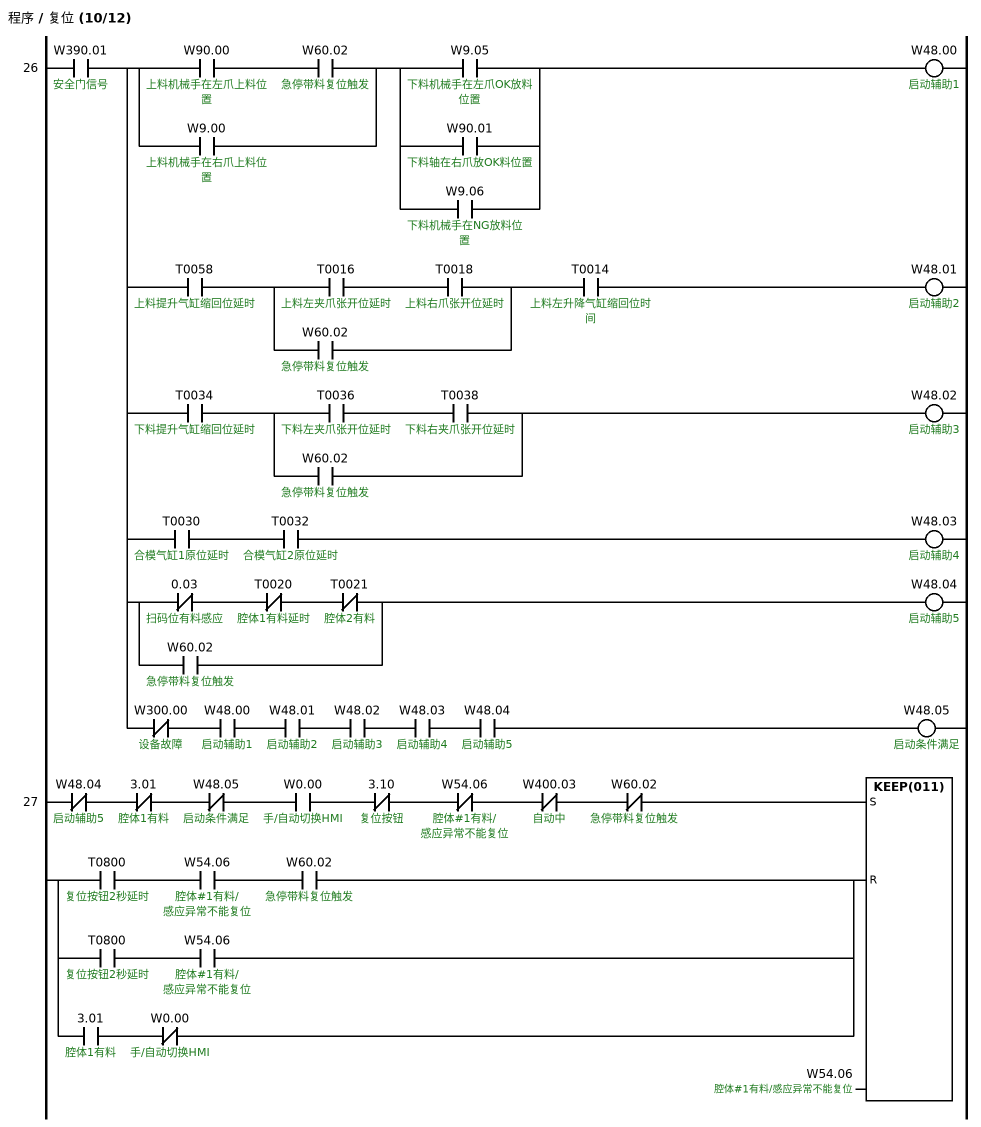
; rung 26
LD W390.01  ; 安全门信号
OUT TR0
LD W90.00  ; 上料机械手在左爪上料位置
AND W60.02  ; 急停带料复位触发
OR W9.00  ; 上料机械手在右爪上料位置
ANDLD
LD W9.05  ; 下料机械手在左爪OK放料位置
OR W90.01  ; 下料轴在右爪放OK料位置
OR W9.06  ; 下料机械手在NG放料位置
ANDLD
OUT W48.00  ; 启动辅助1
LD TR0
AND T0058  ; 上料提升气缸缩回位延时
LD T0016  ; 上料左夹爪张开位延时
AND T0018  ; 上料右爪张开位延时
OR W60.02  ; 急停带料复位触发
ANDLD
AND T0014  ; 上料左升降气缸缩回位时间
OUT W48.01  ; 启动辅助2
LD TR0
AND T0034  ; 下料提升气缸缩回位延时
LD T0036  ; 下料左夹爪张开位延时
AND T0038  ; 下料右夹爪张开位延时
OR W60.02  ; 急停带料复位触发
ANDLD
OUT W48.02  ; 启动辅助3
LD TR0
AND T0030  ; 合模气缸1原位延时
AND T0032  ; 合模气缸2原位延时
OUT W48.03  ; 启动辅助4
LD TR0
LDNOT 0.03  ; 扫码位有料感应
ANDNOT T0020  ; 腔体1有料延时
ANDNOT T0021  ; 腔体2有料
OR W60.02  ; 急停带料复位触发
ANDLD
OUT W48.04  ; 启动辅助5
LD TR0
ANDNOT W300.00  ; 设备故障
AND W48.00  ; 启动辅助1
AND W48.01  ; 启动辅助2
AND W48.02  ; 启动辅助3
AND W48.03  ; 启动辅助4
AND W48.04  ; 启动辅助5
OUT W48.05  ; 启动条件满足
; rung 27
LDNOT W48.04  ; 启动辅助5
ANDNOT 3.01  ; 腔体1有料
ANDNOT W48.05  ; 启动条件满足
AND W0.00  ; 手/自动切换HMI
ANDNOT 3.10  ; 复位按钮
ANDNOT W54.06  ; 腔体#1有料/感应异常不能复位
ANDNOT W400.03  ; 自动中
ANDNOT W60.02  ; 急停带料复位触发
LD T0800  ; 复位按钮2秒延时
AND W54.06  ; 腔体#1有料/感应异常不能复位
AND W60.02  ; 急停带料复位触发
LD T0800  ; 复位按钮2秒延时
AND W54.06  ; 腔体#1有料/感应异常不能复位
ORLD
LD 3.01  ; 腔体1有料
ANDNOT W0.00  ; 手/自动切换HMI
ORLD
KEEP(011) W54.06  ; 腔体#1有料/感应异常不能复位

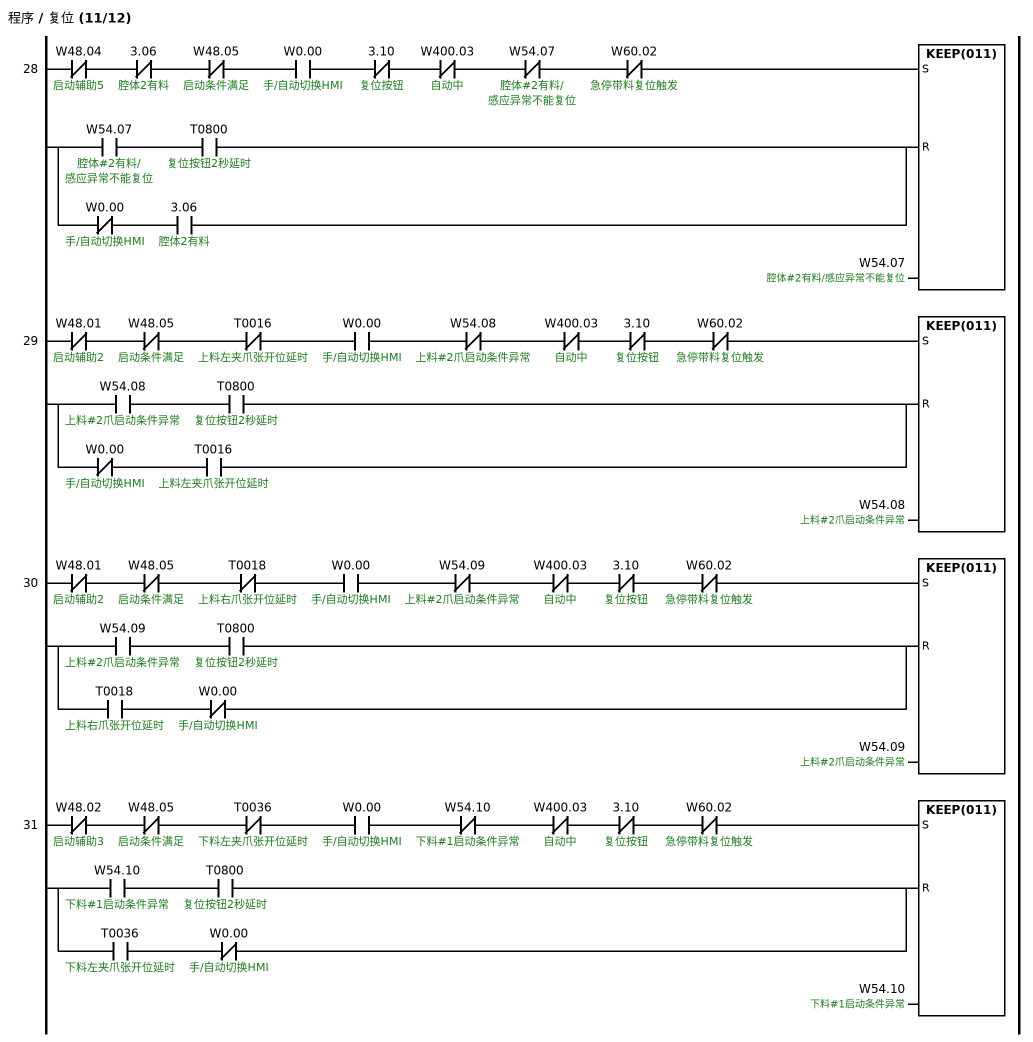
; rung 28
LDNOT W48.04  ; 启动辅助5
ANDNOT 3.06  ; 腔体2有料
ANDNOT W48.05  ; 启动条件满足
AND W0.00  ; 手/自动切换HMI
ANDNOT 3.10  ; 复位按钮
ANDNOT W400.03  ; 自动中
ANDNOT W54.07  ; 腔体#2有料/感应异常不能复位
ANDNOT W60.02  ; 急停带料复位触发
LD W54.07  ; 腔体#2有料/感应异常不能复位
AND T0800  ; 复位按钮2秒延时
LDNOT W0.00  ; 手/自动切换HMI
AND 3.06  ; 腔体2有料
ORLD
KEEP(011) W54.07  ; 腔体#2有料/感应异常不能复位
; rung 29
LDNOT W48.01  ; 启动辅助2
ANDNOT W48.05  ; 启动条件满足
ANDNOT T0016  ; 上料左夹爪张开位延时
AND W0.00  ; 手/自动切换HMI
ANDNOT W54.08  ; 上料#2爪启动条件异常
ANDNOT W400.03  ; 自动中
ANDNOT 3.10  ; 复位按钮
ANDNOT W60.02  ; 急停带料复位触发
LD W54.08  ; 上料#2爪启动条件异常
AND T0800  ; 复位按钮2秒延时
LDNOT W0.00  ; 手/自动切换HMI
AND T0016  ; 上料左夹爪张开位延时
ORLD
KEEP(011) W54.08  ; 上料#2爪启动条件异常
; rung 30
LDNOT W48.01  ; 启动辅助2
ANDNOT W48.05  ; 启动条件满足
ANDNOT T0018  ; 上料右爪张开位延时
AND W0.00  ; 手/自动切换HMI
ANDNOT W54.09  ; 上料#2爪启动条件异常
ANDNOT W400.03  ; 自动中
ANDNOT 3.10  ; 复位按钮
ANDNOT W60.02  ; 急停带料复位触发
LD W54.09  ; 上料#2爪启动条件异常
AND T0800  ; 复位按钮2秒延时
LD T0018  ; 上料右爪张开位延时
ANDNOT W0.00  ; 手/自动切换HMI
ORLD
KEEP(011) W54.09  ; 上料#2爪启动条件异常
; rung 31
LDNOT W48.02  ; 启动辅助3
ANDNOT W48.05  ; 启动条件满足
ANDNOT T0036  ; 下料左夹爪张开位延时
AND W0.00  ; 手/自动切换HMI
ANDNOT W54.10  ; 下料#1启动条件异常
ANDNOT W400.03  ; 自动中
ANDNOT 3.10  ; 复位按钮
ANDNOT W60.02  ; 急停带料复位触发
LD W54.10  ; 下料#1启动条件异常
AND T0800  ; 复位按钮2秒延时
LD T0036  ; 下料左夹爪张开位延时
ANDNOT W0.00  ; 手/自动切换HMI
ORLD
KEEP(011) W54.10  ; 下料#1启动条件异常

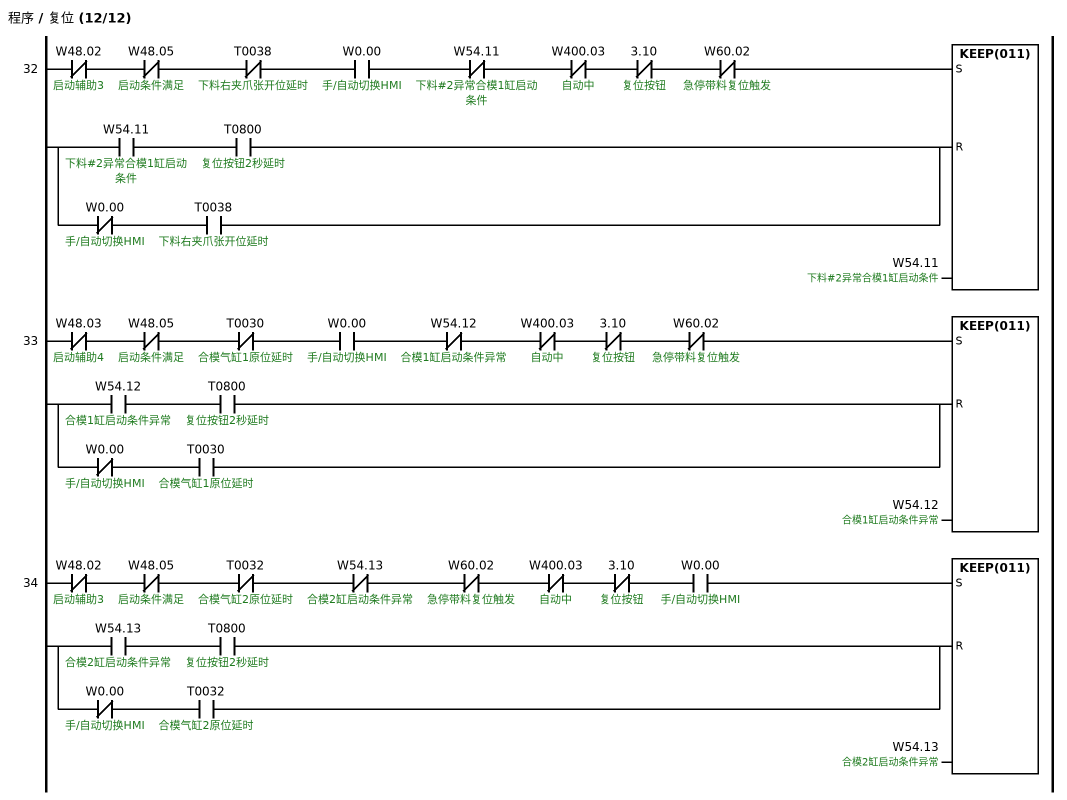
; rung 32
LDNOT W48.02  ; 启动辅助3
ANDNOT W48.05  ; 启动条件满足
ANDNOT T0038  ; 下料右夹爪张开位延时
AND W0.00  ; 手/自动切换HMI
ANDNOT W54.11  ; 下料#2异常合模1缸启动条件
ANDNOT W400.03  ; 自动中
ANDNOT 3.10  ; 复位按钮
ANDNOT W60.02  ; 急停带料复位触发
LD W54.11  ; 下料#2异常合模1缸启动条件
AND T0800  ; 复位按钮2秒延时
LDNOT W0.00  ; 手/自动切换HMI
AND T0038  ; 下料右夹爪张开位延时
ORLD
KEEP(011) W54.11  ; 下料#2异常合模1缸启动条件
; rung 33
LDNOT W48.03  ; 启动辅助4
ANDNOT W48.05  ; 启动条件满足
ANDNOT T0030  ; 合模气缸1原位延时
AND W0.00  ; 手/自动切换HMI
ANDNOT W54.12  ; 合模1缸启动条件异常
ANDNOT W400.03  ; 自动中
ANDNOT 3.10  ; 复位按钮
ANDNOT W60.02  ; 急停带料复位触发
LD W54.12  ; 合模1缸启动条件异常
AND T0800  ; 复位按钮2秒延时
LDNOT W0.00  ; 手/自动切换HMI
AND T0030  ; 合模气缸1原位延时
ORLD
KEEP(011) W54.12  ; 合模1缸启动条件异常
; rung 34
LDNOT W48.02  ; 启动辅助3
ANDNOT W48.05  ; 启动条件满足
ANDNOT T0032  ; 合模气缸2原位延时
ANDNOT W54.13  ; 合模2缸启动条件异常
ANDNOT W60.02  ; 急停带料复位触发
ANDNOT W400.03  ; 自动中
ANDNOT 3.10  ; 复位按钮
AND W0.00  ; 手/自动切换HMI
LD W54.13  ; 合模2缸启动条件异常
AND T0800  ; 复位按钮2秒延时
LDNOT W0.00  ; 手/自动切换HMI
AND T0032  ; 合模气缸2原位延时
ORLD
KEEP(011) W54.13  ; 合模2缸启动条件异常

### Section 条码读取（模1端1）

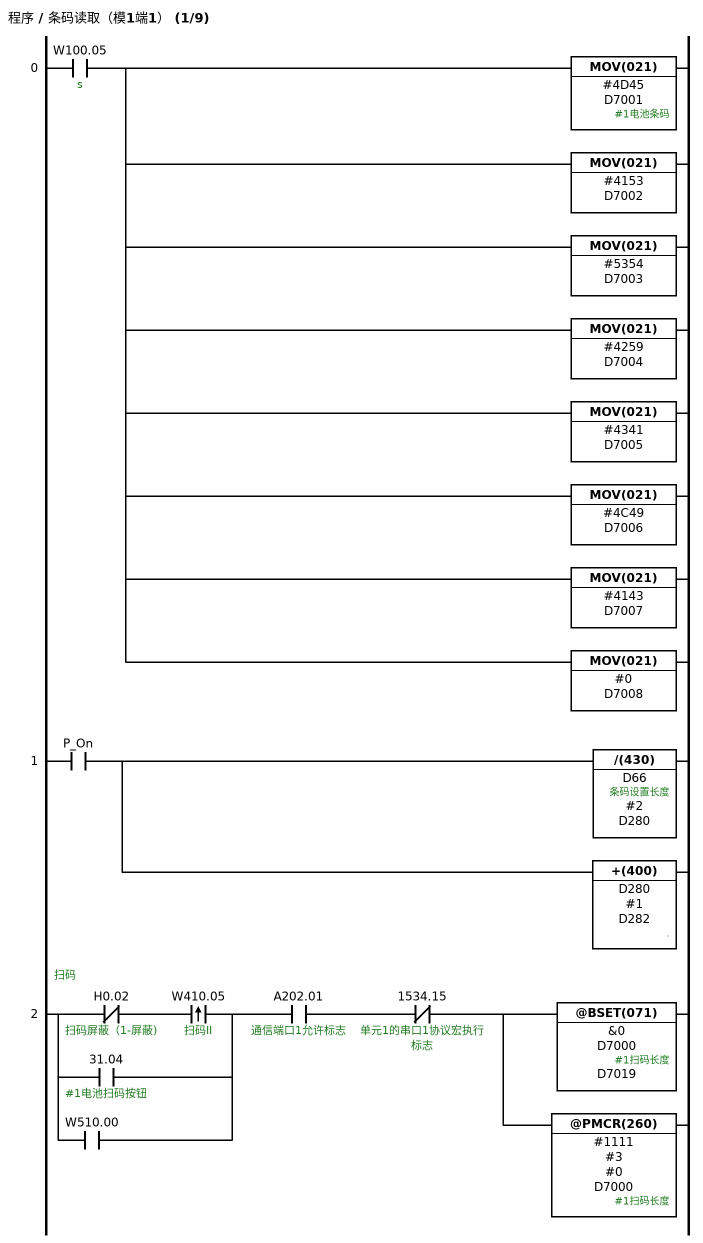
; rung 0
LD W100.05  ; s
MOV(021) #4D45 D7001  ; #1电池条码
MOV(021) #4153 D7002
MOV(021) #5354 D7003
MOV(021) #4259 D7004
MOV(021) #4341 D7005
MOV(021) #4C49 D7006
MOV(021) #4143 D7007
MOV(021) #0 D7008
; rung 1
LD P_On
/(430) D66 #2 D280  ; 条码设置长度
+(400) D280 #1 D282  ; .
; rung 2: 扫码
LDNOT H0.02  ; 扫码屏蔽（1-屏蔽)
@AND W410.05  ; 扫码II
OR 31.04  ; #1电池扫码按钮
OR W510.00
AND A202.01  ; 通信端口1允许标志
ANDNOT 1534.15  ; 单元1的串口1协议宏执行标志
@BSET(071) &0 D7000 D7019  ; #1扫码长度
@PMCR(260) #1111 #3 #0 D7000  ; #1扫码长度

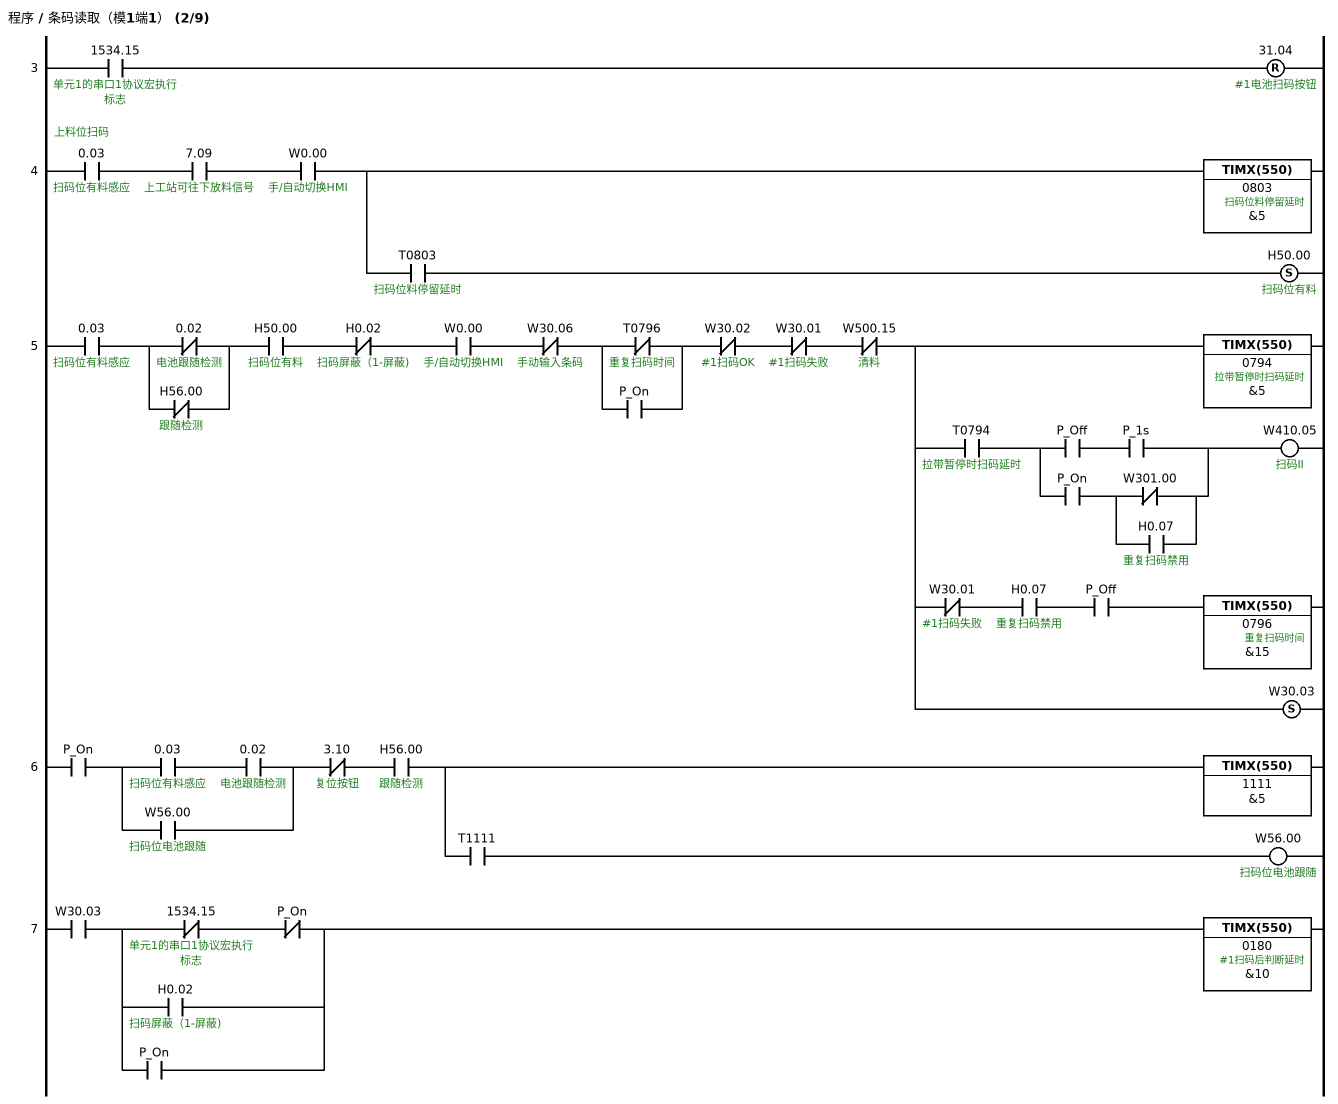
; rung 3
LD 1534.15  ; 单元1的串口1协议宏执行标志
RSET 31.04  ; #1电池扫码按钮
; rung 4: 上料位扫码
LD 0.03  ; 扫码位有料感应
AND 7.09  ; 上工站可往下放料信号
AND W0.00  ; 手/自动切换HMI
TIMX(550) 0803 &5  ; 扫码位料停留延时
AND T0803  ; 扫码位料停留延时
SET H50.00  ; 扫码位有料
; rung 5
LD 0.03  ; 扫码位有料感应
LDNOT 0.02  ; 电池跟随检测
ORNOT H56.00  ; 跟随检测
ANDLD
AND H50.00  ; 扫码位有料
ANDNOT H0.02  ; 扫码屏蔽（1-屏蔽)
AND W0.00  ; 手/自动切换HMI
ANDNOT W30.06  ; 手动输入条码
LDNOT T0796  ; 重复扫码时间
OR P_On
ANDLD
ANDNOT W30.02  ; #1扫码OK
ANDNOT W30.01  ; #1扫码失败
ANDNOT W500.15  ; 清料
OUT TR0
TIMX(550) 0794 &5  ; 拉带暂停时扫码延时
AND T0794  ; 拉带暂停时扫码延时
LD P_Off
AND P_1s
LD P_On
LDNOT W301.00
OR H0.07  ; 重复扫码禁用
ANDLD
ORLD
ANDLD
OUT W410.05  ; 扫码II
LD TR0
ANDNOT W30.01  ; #1扫码失败
AND H0.07  ; 重复扫码禁用
AND P_Off
TIMX(550) 0796 &15  ; 重复扫码时间
LD TR0
SET W30.03
; rung 6
LD P_On
LD 0.03  ; 扫码位有料感应
AND 0.02  ; 电池跟随检测
OR W56.00  ; 扫码位电池跟随
ANDLD
ANDNOT 3.10  ; 复位按钮
AND H56.00  ; 跟随检测
TIMX(550) 1111 &5
AND T1111
OUT W56.00  ; 扫码位电池跟随
; rung 7
LD W30.03
LDNOT 1534.15  ; 单元1的串口1协议宏执行标志
ANDNOT P_On
OR H0.02  ; 扫码屏蔽（1-屏蔽)
OR P_On
ANDLD
TIMX(550) 0180 &10  ; #1扫码后判断延时

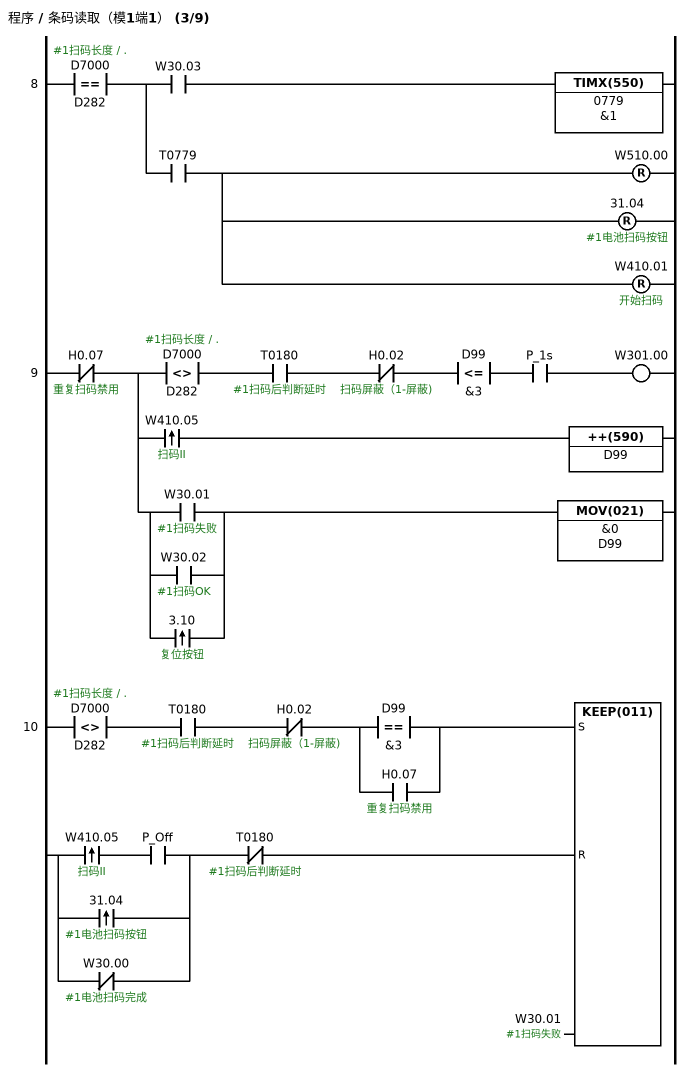
; rung 8
LD=(300) D7000 D282  ; #1扫码长度, .
OUT TR0
AND W30.03
TIMX(550) 0779 &1
LD TR0
AND T0779
RSET W510.00
RSET 31.04  ; #1电池扫码按钮
RSET W410.01  ; 开始扫码
; rung 9
LDNOT H0.07  ; 重复扫码禁用
OUT TR0
AND<>(305) D7000 D282  ; #1扫码长度, .
AND T0180  ; #1扫码后判断延时
ANDNOT H0.02  ; 扫码屏蔽（1-屏蔽)
AND<=(315) D99 &3
AND P_1s
OUT W301.00
LD TR0
@AND W410.05  ; 扫码II
++(590) D99
LD TR0
LD W30.01  ; #1扫码失败
OR W30.02  ; #1扫码OK
@OR 3.10  ; 复位按钮
ANDLD
MOV(021) &0 D99
; rung 10
LD<>(305) D7000 D282  ; #1扫码长度, .
AND T0180  ; #1扫码后判断延时
ANDNOT H0.02  ; 扫码屏蔽（1-屏蔽)
LD=(300) D99 &3
OR H0.07  ; 重复扫码禁用
ANDLD
@LD W410.05  ; 扫码II
AND P_Off
@OR 31.04  ; #1电池扫码按钮
ORNOT W30.00  ; #1电池扫码完成
ANDNOT T0180  ; #1扫码后判断延时
KEEP(011) W30.01  ; #1扫码失败

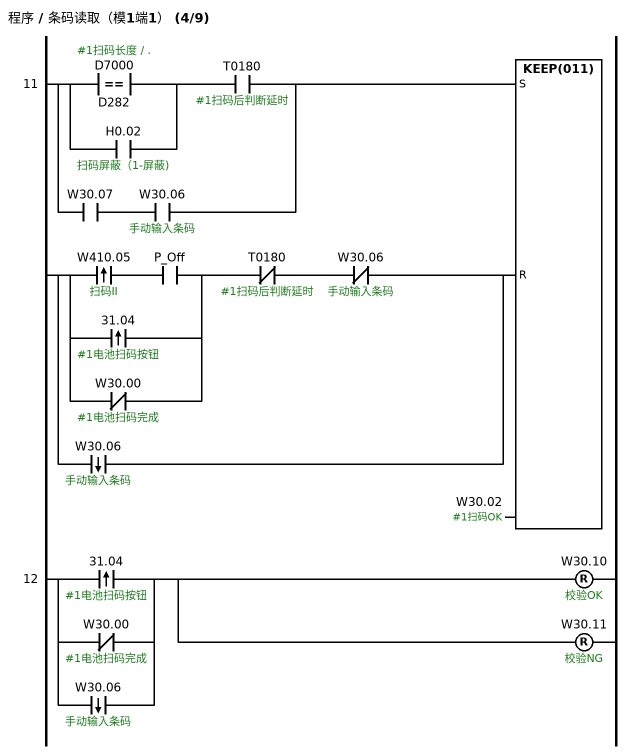
; rung 11
LD=(300) D7000 D282  ; #1扫码长度, .
OR H0.02  ; 扫码屏蔽（1-屏蔽)
AND T0180  ; #1扫码后判断延时
LD W30.07
AND W30.06  ; 手动输入条码
ORLD
@LD W410.05  ; 扫码II
AND P_Off
@OR 31.04  ; #1电池扫码按钮
ORNOT W30.00  ; #1电池扫码完成
ANDNOT T0180  ; #1扫码后判断延时
ANDNOT W30.06  ; 手动输入条码
%OR W30.06  ; 手动输入条码
KEEP(011) W30.02  ; #1扫码OK
; rung 12
@LD 31.04  ; #1电池扫码按钮
ORNOT W30.00  ; #1电池扫码完成
%OR W30.06  ; 手动输入条码
RSET W30.10  ; 校验OK
RSET W30.11  ; 校验NG

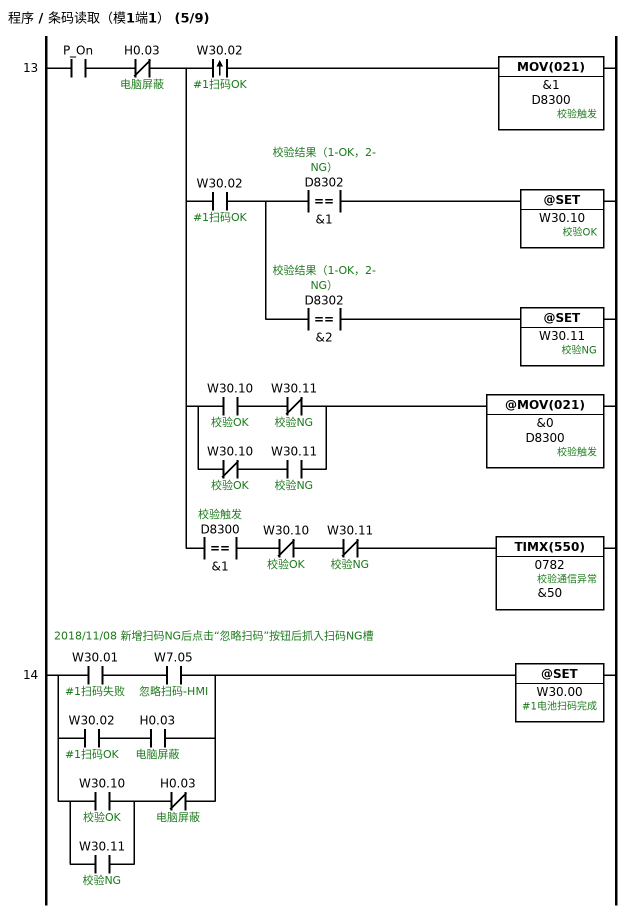
; rung 13
LD P_On
ANDNOT H0.03  ; 电脑屏蔽
OUT TR0
@AND W30.02  ; #1扫码OK
MOV(021) &1 D8300  ; 校验触发
LD TR0
AND W30.02  ; #1扫码OK
OUT TR1
AND=(300) D8302 &1  ; 校验结果（1-OK，2-NG）
@SET W30.10  ; 校验OK
LD TR1
AND=(300) D8302 &2  ; 校验结果（1-OK，2-NG）
@SET W30.11  ; 校验NG
LD TR0
LD W30.10  ; 校验OK
ANDNOT W30.11  ; 校验NG
LDNOT W30.10  ; 校验OK
AND W30.11  ; 校验NG
ORLD
ANDLD
@MOV(021) &0 D8300  ; 校验触发
LD TR0
AND=(300) D8300 &1  ; 校验触发
ANDNOT W30.10  ; 校验OK
ANDNOT W30.11  ; 校验NG
TIMX(550) 0782 &50  ; 校验通信异常
; rung 14: 2018/11/08 新增扫码NG后点击“忽略扫码”按钮后抓入扫码NG槽
LD W30.01  ; #1扫码失败
AND W7.05  ; 忽略扫码-HMI  // 新增扫码NG后点击“忽略扫码”后抓入扫码NG槽
LD W30.02  ; #1扫码OK
AND H0.03  ; 电脑屏蔽
ORLD
LD W30.10  ; 校验OK
OR W30.11  ; 校验NG
ANDNOT H0.03  ; 电脑屏蔽
ORLD
@SET W30.00  ; #1电池扫码完成

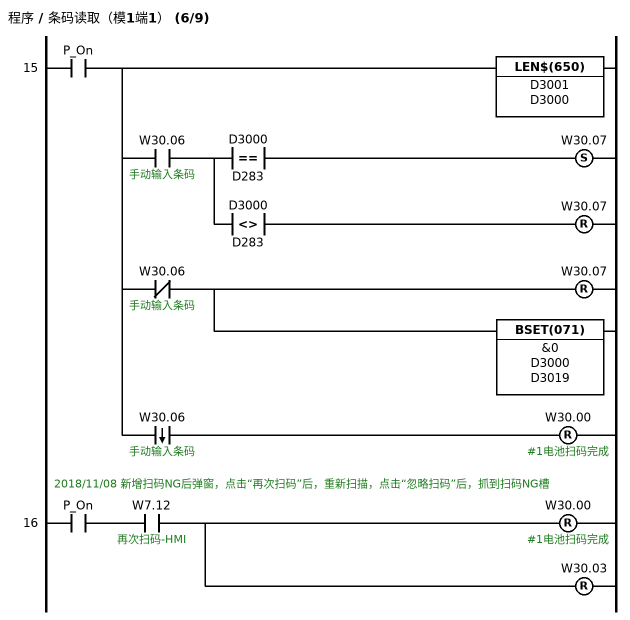
; rung 15
LD P_On
OUT TR0
LEN$(650) D3001 D3000
AND W30.06  ; 手动输入条码
OUT TR1
AND=(300) D3000 D283
SET W30.07
LD TR1
AND<>(305) D3000 D283
RSET W30.07
LD TR0
ANDNOT W30.06  ; 手动输入条码
RSET W30.07
BSET(071) &0 D3000 D3019
LD TR0
%AND W30.06  ; 手动输入条码
RSET W30.00  ; #1电池扫码完成
; rung 16: 2018/11/08 新增扫码NG后弹窗，点击“再次扫码”后，重新扫描，点击“忽略扫码”后，抓到扫码NG槽
LD P_On
AND W7.12  ; 再次扫码-HMI
RSET W30.00  ; #1电池扫码完成
RSET W30.03

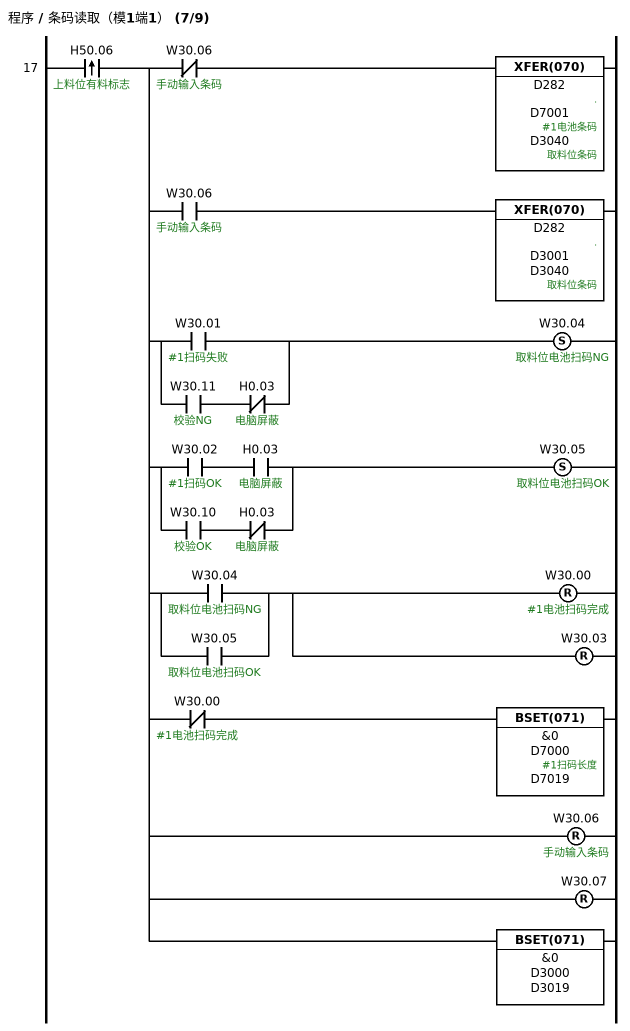
; rung 17
@LD H50.06  ; 上料位有料标志
OUT TR0
ANDNOT W30.06  ; 手动输入条码
XFER(070) D282 D7001 D3040  ; ., #1电池条码, 取料位条码
LD TR0
AND W30.06  ; 手动输入条码
XFER(070) D282 D3001 D3040  ; ., 取料位条码
LD TR0
LD W30.01  ; #1扫码失败
LD W30.11  ; 校验NG
ANDNOT H0.03  ; 电脑屏蔽
ORLD
ANDLD
SET W30.04  ; 取料位电池扫码NG
LD TR0
LD W30.02  ; #1扫码OK
AND H0.03  ; 电脑屏蔽
LD W30.10  ; 校验OK
ANDNOT H0.03  ; 电脑屏蔽
ORLD
ANDLD
SET W30.05  ; 取料位电池扫码OK
LD TR0
LD W30.04  ; 取料位电池扫码NG
OR W30.05  ; 取料位电池扫码OK
ANDLD
RSET W30.00  ; #1电池扫码完成
RSET W30.03
LD TR0
ANDNOT W30.00  ; #1电池扫码完成
BSET(071) &0 D7000 D7019  ; #1扫码长度
LD TR0
RSET W30.06  ; 手动输入条码
RSET W30.07
BSET(071) &0 D3000 D3019

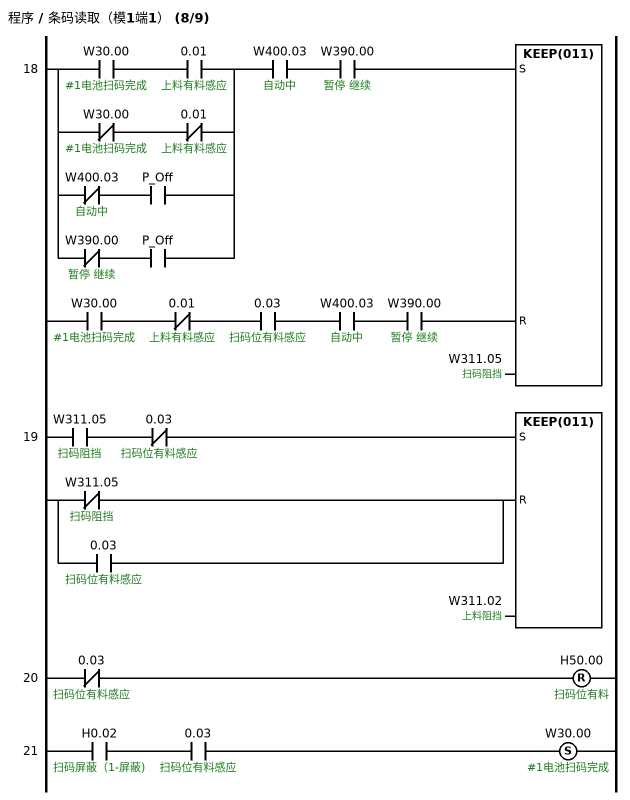
; rung 18
LD W30.00  ; #1电池扫码完成
AND 0.01  ; 上料有料感应
LDNOT W30.00  ; #1电池扫码完成
ANDNOT 0.01  ; 上料有料感应
ORLD
LDNOT W400.03  ; 自动中
AND P_Off
ORLD
LDNOT W390.00  ; 暂停 继续
AND P_Off
ORLD
AND W400.03  ; 自动中
AND W390.00  ; 暂停 继续
LD W30.00  ; #1电池扫码完成
ANDNOT 0.01  ; 上料有料感应
AND 0.03  ; 扫码位有料感应
AND W400.03  ; 自动中
AND W390.00  ; 暂停 继续
KEEP(011) W311.05  ; 扫码阻挡
; rung 19
LD W311.05  ; 扫码阻挡
ANDNOT 0.03  ; 扫码位有料感应
LDNOT W311.05  ; 扫码阻挡
OR 0.03  ; 扫码位有料感应
KEEP(011) W311.02  ; 上料阻挡
; rung 20
LDNOT 0.03  ; 扫码位有料感应
RSET H50.00  ; 扫码位有料
; rung 21
LD H0.02  ; 扫码屏蔽（1-屏蔽)
AND 0.03  ; 扫码位有料感应
SET W30.00  ; #1电池扫码完成

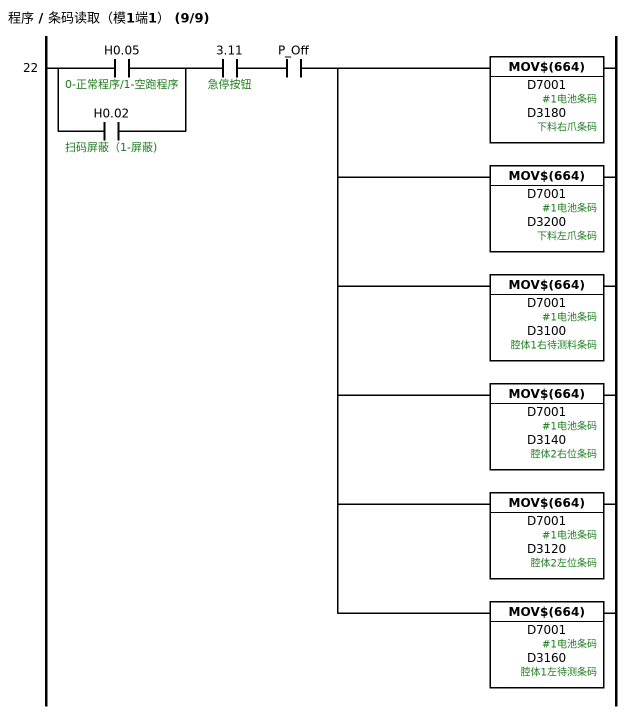
; rung 22
LD H0.05  ; 0-正常程序/1-空跑程序
OR H0.02  ; 扫码屏蔽（1-屏蔽)
AND 3.11  ; 急停按钮
AND P_Off
MOV$(664) D7001 D3180  ; #1电池条码, 下料右爪条码
MOV$(664) D7001 D3200  ; #1电池条码, 下料左爪条码
MOV$(664) D7001 D3100  ; #1电池条码, 腔体1右待测料条码
MOV$(664) D7001 D3140  ; #1电池条码, 腔体2右位条码
MOV$(664) D7001 D3120  ; #1电池条码, 腔体2左位条码
MOV$(664) D7001 D3160  ; #1电池条码, 腔体1左待测条码

### Section 上料轴自动

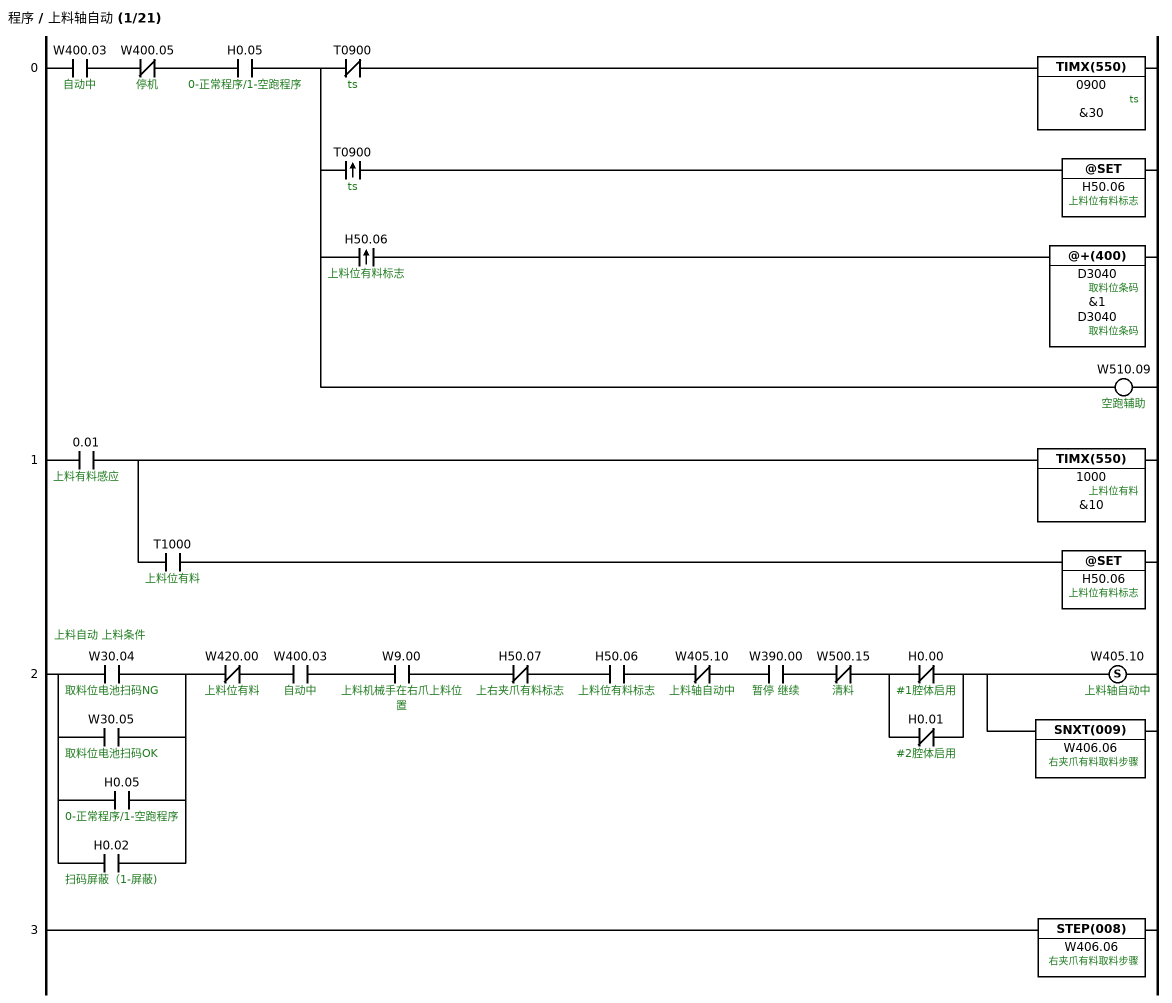
; rung 0
LD W400.03  ; 自动中
ANDNOT W400.05  ; 停机
AND H0.05  ; 0-正常程序/1-空跑程序
OUT TR0
ANDNOT T0900  ; ts
TIMX(550) 0900 &30  ; ts
LD TR0
@AND T0900  ; ts
@SET H50.06  ; 上料位有料标志
LD TR0
@AND H50.06  ; 上料位有料标志
@+(400) D3040 &1 D3040  ; 取料位条码
LD TR0
OUT W510.09  ; 空跑辅助
; rung 1
LD 0.01  ; 上料有料感应
TIMX(550) 1000 &10  ; 上料位有料
AND T1000  ; 上料位有料
@SET H50.06  ; 上料位有料标志
; rung 2: 上料自动 上料条件
LD W30.04  ; 取料位电池扫码NG
OR W30.05  ; 取料位电池扫码OK
OR H0.05  ; 0-正常程序/1-空跑程序
OR H0.02  ; 扫码屏蔽（1-屏蔽)
ANDNOT W420.00  ; 上料位有料
AND W400.03  ; 自动中
AND W9.00  ; 上料机械手在右爪上料位置
ANDNOT H50.07  ; 上右夹爪有料标志
AND H50.06  ; 上料位有料标志
ANDNOT W405.10  ; 上料轴自动中
AND W390.00  ; 暂停 继续
ANDNOT W500.15  ; 清料
LDNOT H0.00  ; #1腔体启用
ORNOT H0.01  ; #2腔体启用
ANDLD
SET W405.10  ; 上料轴自动中
SNXT(009) W406.06  ; 右夹爪有料取料步骤
; rung 3
STEP(008) W406.06  ; 右夹爪有料取料步骤

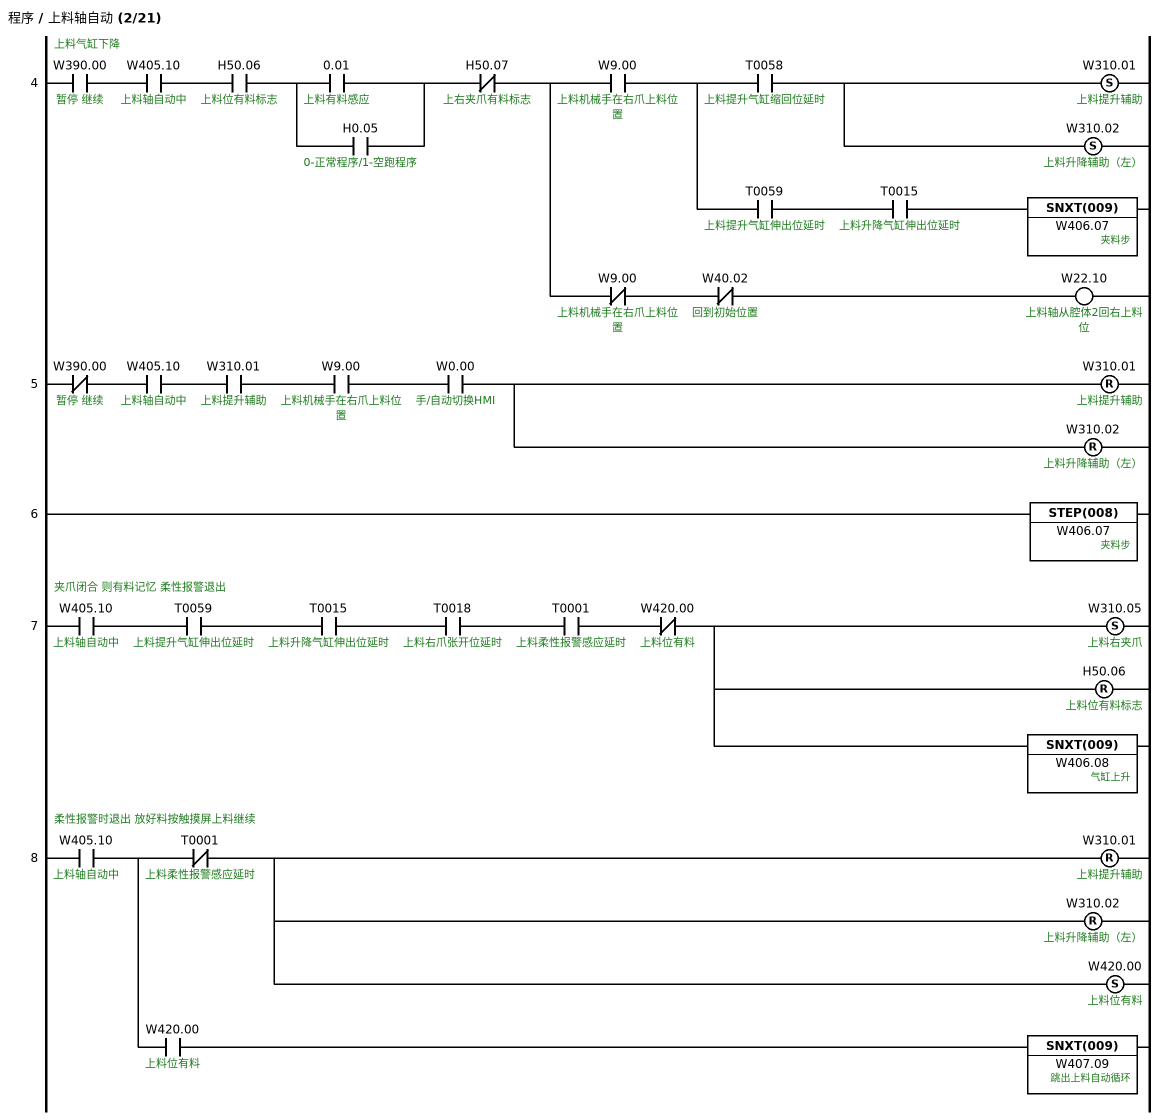
; rung 4: 上料气缸下降
LD W390.00  ; 暂停 继续
AND W405.10  ; 上料轴自动中
AND H50.06  ; 上料位有料标志
LD 0.01  ; 上料有料感应
OR H0.05  ; 0-正常程序/1-空跑程序
ANDLD
ANDNOT H50.07  ; 上右夹爪有料标志
OUT TR0
AND W9.00  ; 上料机械手在右爪上料位置
OUT TR1
AND T0058  ; 上料提升气缸缩回位延时
SET W310.01  ; 上料提升辅助
SET W310.02  ; 上料升降辅助（左）
LD TR1
AND T0059  ; 上料提升气缸伸出位延时
AND T0015  ; 上料升降气缸伸出位延时
SNXT(009) W406.07  ; 夹料步
LD TR0
ANDNOT W9.00  ; 上料机械手在右爪上料位置
ANDNOT W40.02  ; 回到初始位置
OUT W22.10  ; 上料轴从腔体2回右上料位
; rung 5
LDNOT W390.00  ; 暂停 继续
AND W405.10  ; 上料轴自动中
AND W310.01  ; 上料提升辅助
AND W9.00  ; 上料机械手在右爪上料位置
AND W0.00  ; 手/自动切换HMI
RSET W310.01  ; 上料提升辅助
RSET W310.02  ; 上料升降辅助（左）
; rung 6
STEP(008) W406.07  ; 夹料步
; rung 7: 夹爪闭合 则有料记忆 柔性报警退出
LD W405.10  ; 上料轴自动中
AND T0059  ; 上料提升气缸伸出位延时
AND T0015  ; 上料升降气缸伸出位延时
AND T0018  ; 上料右爪张开位延时
AND T0001  ; 上料柔性报警感应延时
ANDNOT W420.00  ; 上料位有料
SET W310.05  ; 上料右夹爪
RSET H50.06  ; 上料位有料标志
SNXT(009) W406.08  ; 气缸上升
; rung 8: 柔性报警时退出 放好料按触摸屏上料继续
LD W405.10  ; 上料轴自动中
OUT TR0
ANDNOT T0001  ; 上料柔性报警感应延时
RSET W310.01  ; 上料提升辅助
RSET W310.02  ; 上料升降辅助（左）
SET W420.00  ; 上料位有料
LD TR0
AND W420.00  ; 上料位有料
SNXT(009) W407.09  ; 跳出上料自动循环

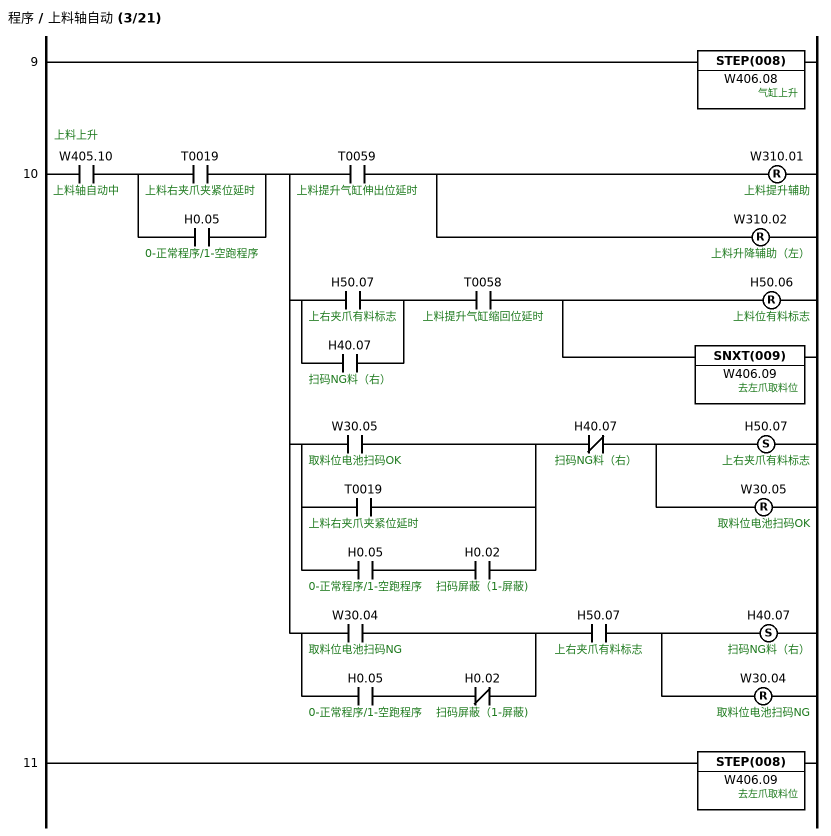
; rung 9
STEP(008) W406.08  ; 气缸上升
; rung 10: 上料上升
LD W405.10  ; 上料轴自动中
LD T0019  ; 上料右夹爪夹紧位延时
OR H0.05  ; 0-正常程序/1-空跑程序
ANDLD
OUT TR0
AND T0059  ; 上料提升气缸伸出位延时
RSET W310.01  ; 上料提升辅助
RSET W310.02  ; 上料升降辅助（左）
LD TR0
LD H50.07  ; 上右夹爪有料标志
OR H40.07  ; 扫码NG料（右）
ANDLD
AND T0058  ; 上料提升气缸缩回位延时
RSET H50.06  ; 上料位有料标志
SNXT(009) W406.09  ; 去左爪取料位
LD TR0
LD W30.05  ; 取料位电池扫码OK
OR T0019  ; 上料右夹爪夹紧位延时
LD H0.05  ; 0-正常程序/1-空跑程序
AND H0.02  ; 扫码屏蔽（1-屏蔽)
ORLD
ANDLD
ANDNOT H40.07  ; 扫码NG料（右）
SET H50.07  ; 上右夹爪有料标志
RSET W30.05  ; 取料位电池扫码OK
LD TR0
LD W30.04  ; 取料位电池扫码NG
LD H0.05  ; 0-正常程序/1-空跑程序
ANDNOT H0.02  ; 扫码屏蔽（1-屏蔽)
ORLD
ANDLD
AND H50.07  ; 上右夹爪有料标志
SET H40.07  ; 扫码NG料（右）
RSET W30.04  ; 取料位电池扫码NG
; rung 11
STEP(008) W406.09  ; 去左爪取料位

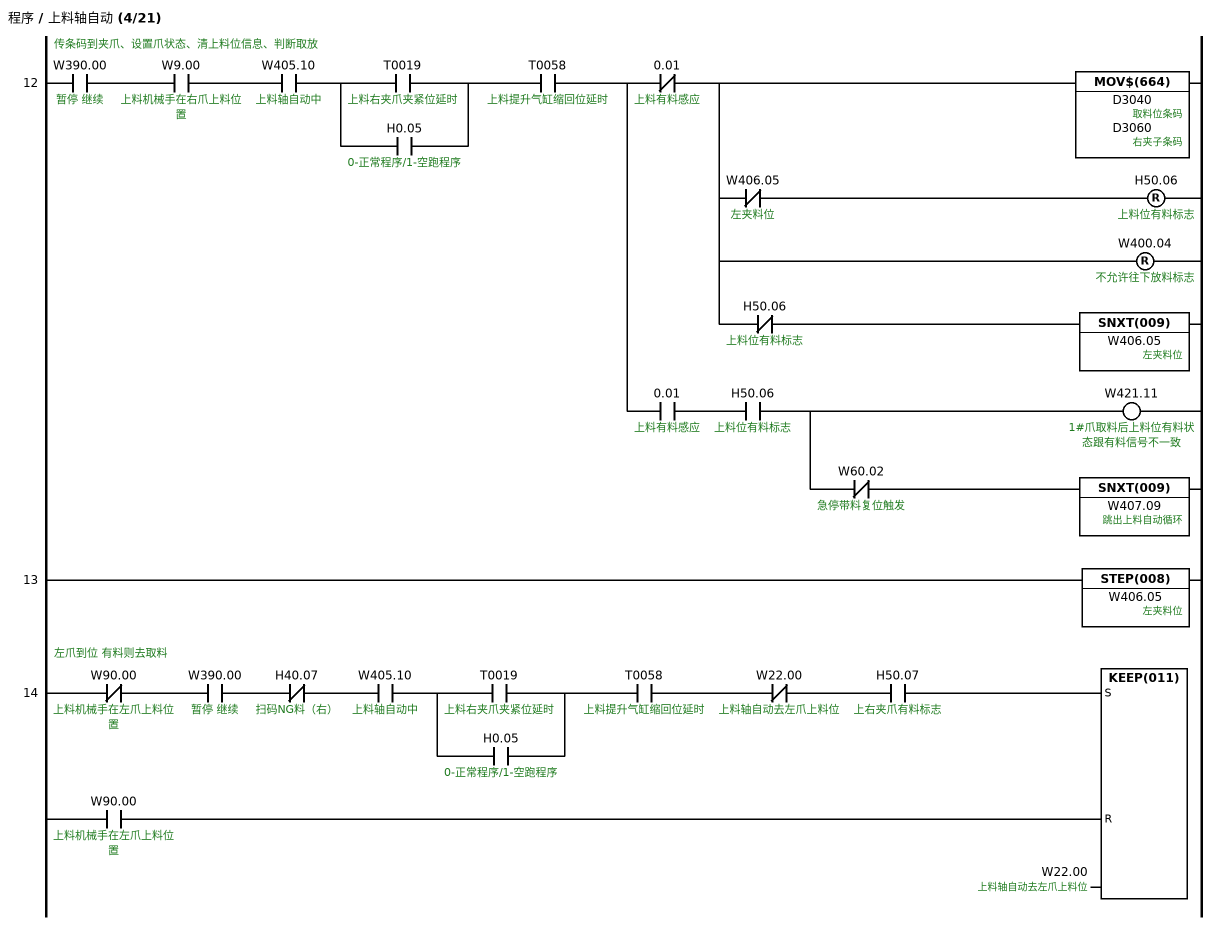
; rung 12: 传条码到夹爪、设置爪状态、清上料位信息、判断取放
LD W390.00  ; 暂停 继续
AND W9.00  ; 上料机械手在右爪上料位置
AND W405.10  ; 上料轴自动中
LD T0019  ; 上料右夹爪夹紧位延时
OR H0.05  ; 0-正常程序/1-空跑程序
ANDLD
AND T0058  ; 上料提升气缸缩回位延时
OUT TR0
ANDNOT 0.01  ; 上料有料感应
OUT TR1
MOV$(664) D3040 D3060  ; 取料位条码, 右夹子条码
ANDNOT W406.05  ; 左夹料位
RSET H50.06  ; 上料位有料标志
LD TR1
RSET W400.04  ; 不允许往下放料标志
ANDNOT H50.06  ; 上料位有料标志
SNXT(009) W406.05  ; 左夹料位
LD TR0
AND 0.01  ; 上料有料感应
AND H50.06  ; 上料位有料标志
OUT W421.11  ; 1#爪取料后上料位有料状态跟有料信号不一致
ANDNOT W60.02  ; 急停带料复位触发
SNXT(009) W407.09  ; 跳出上料自动循环
; rung 13
STEP(008) W406.05  ; 左夹料位
; rung 14: 左爪到位 有料则去取料
LDNOT W90.00  ; 上料机械手在左爪上料位置
AND W390.00  ; 暂停 继续
ANDNOT H40.07  ; 扫码NG料（右）
AND W405.10  ; 上料轴自动中
LD T0019  ; 上料右夹爪夹紧位延时
OR H0.05  ; 0-正常程序/1-空跑程序
ANDLD
AND T0058  ; 上料提升气缸缩回位延时
ANDNOT W22.00  ; 上料轴自动去左爪上料位
AND H50.07  ; 上右夹爪有料标志
LD W90.00  ; 上料机械手在左爪上料位置
KEEP(011) W22.00  ; 上料轴自动去左爪上料位

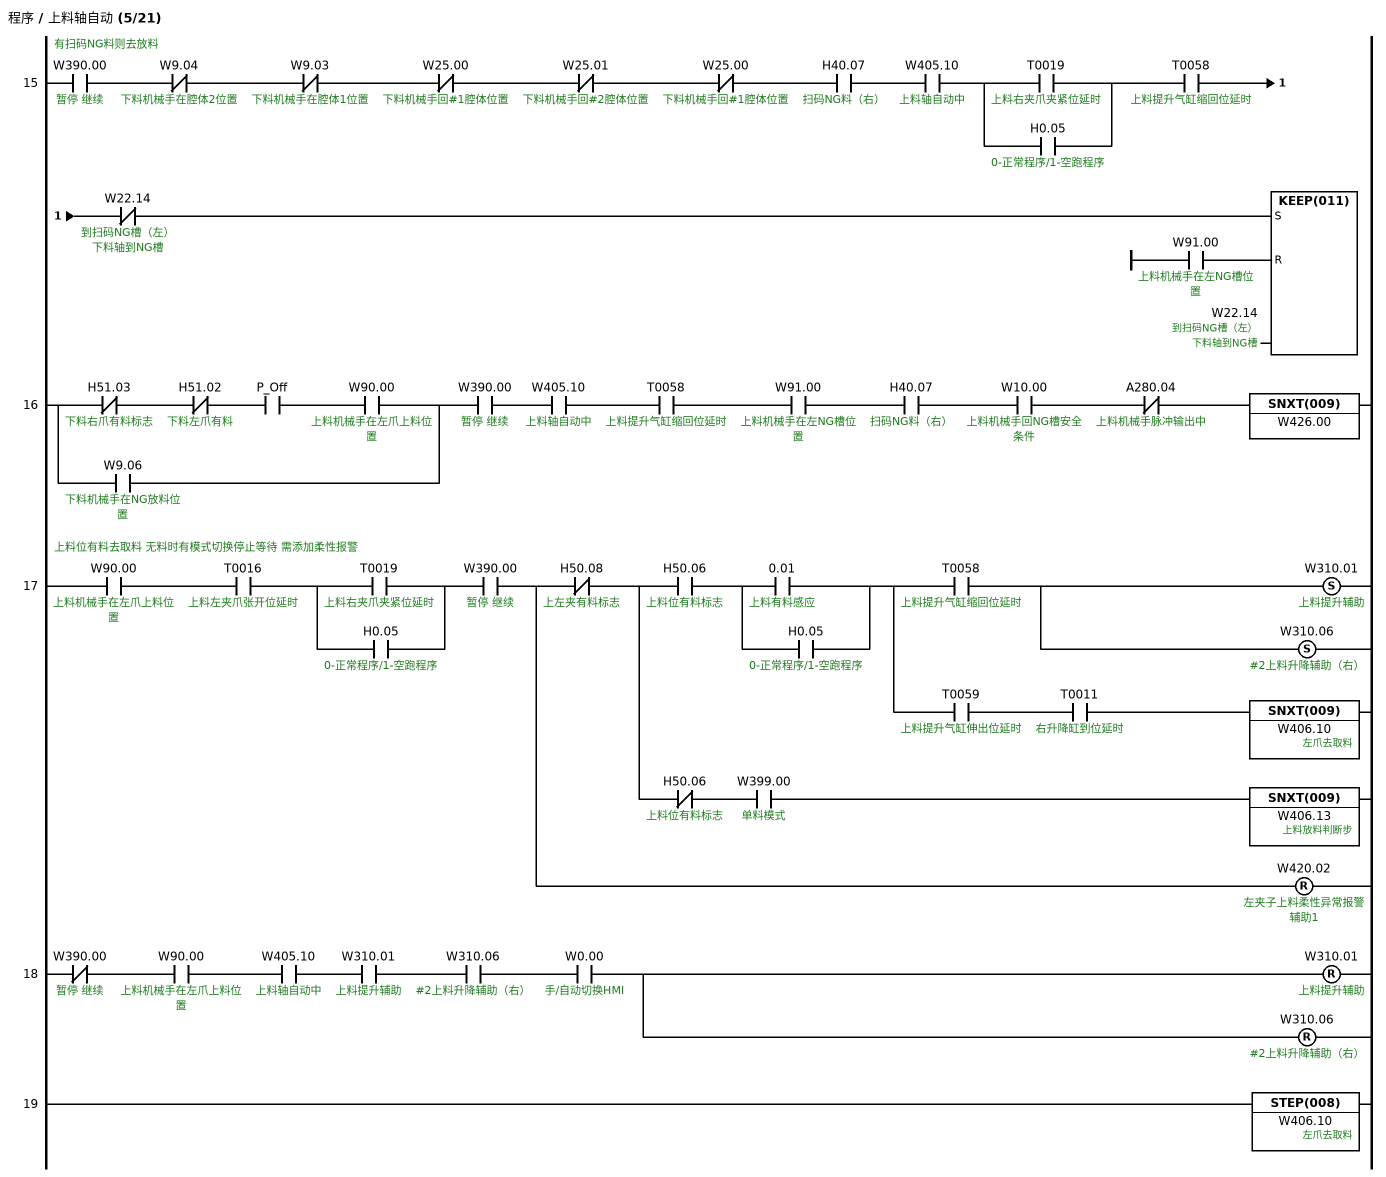
; rung 15: 有扫码NG料则去放料
LD W390.00  ; 暂停 继续
ANDNOT W9.04  ; 下料机械手在腔体2位置
ANDNOT W9.03  ; 下料机械手在腔体1位置
ANDNOT W25.00  ; 下料机械手回#1腔体位置
ANDNOT W25.01  ; 下料机械手回#2腔体位置
ANDNOT W25.00  ; 下料机械手回#1腔体位置
AND H40.07  ; 扫码NG料（右）
AND W405.10  ; 上料轴自动中
LD T0019  ; 上料右夹爪夹紧位延时
OR H0.05  ; 0-正常程序/1-空跑程序
ANDLD
AND T0058  ; 上料提升气缸缩回位延时
ANDNOT W22.14  ; 到扫码NG槽（左） 下料轴到NG槽
LD W91.00  ; 上料机械手在左NG槽位置
KEEP(011) W22.14  ; 到扫码NG槽（左） 下料轴到NG槽
; rung 16
LDNOT H51.03  ; 下料右爪有料标志
ANDNOT H51.02  ; 下料左爪有料
AND P_Off
AND W90.00  ; 上料机械手在左爪上料位置
OR W9.06  ; 下料机械手在NG放料位置
AND W390.00  ; 暂停 继续
AND W405.10  ; 上料轴自动中
AND T0058  ; 上料提升气缸缩回位延时
AND W91.00  ; 上料机械手在左NG槽位置
AND H40.07  ; 扫码NG料（右）
AND W10.00  ; 上料机械手回NG槽安全条件
ANDNOT A280.04  ; 上料机械手脉冲输出中
SNXT(009) W426.00
; rung 17: 上料位有料去取料 无料时有模式切换停止等待 需添加柔性报警
LD W90.00  ; 上料机械手在左爪上料位置
AND T0016  ; 上料左夹爪张开位延时
LD T0019  ; 上料右夹爪夹紧位延时
OR H0.05  ; 0-正常程序/1-空跑程序
ANDLD
AND W390.00  ; 暂停 继续
OUT TR0
ANDNOT H50.08  ; 上左夹有料标志
OUT TR1
AND H50.06  ; 上料位有料标志
LD 0.01  ; 上料有料感应
OR H0.05  ; 0-正常程序/1-空跑程序
ANDLD
OUT TR2
AND T0058  ; 上料提升气缸缩回位延时
SET W310.01  ; 上料提升辅助
SET W310.06  ; #2上料升降辅助（右）
LD TR2
AND T0059  ; 上料提升气缸伸出位延时
AND T0011  ; 右升降缸到位延时
SNXT(009) W406.10  ; 左爪去取料
LD TR1
ANDNOT H50.06  ; 上料位有料标志
AND W399.00  ; 单料模式
SNXT(009) W406.13  ; 上料放料判断步
LD TR0
RSET W420.02  ; 左夹子上料柔性异常报警辅助1
; rung 18
LDNOT W390.00  ; 暂停 继续
AND W90.00  ; 上料机械手在左爪上料位置
AND W405.10  ; 上料轴自动中
AND W310.01  ; 上料提升辅助
AND W310.06  ; #2上料升降辅助（右）
AND W0.00  ; 手/自动切换HMI
RSET W310.01  ; 上料提升辅助
RSET W310.06  ; #2上料升降辅助（右）
; rung 19
STEP(008) W406.10  ; 左爪去取料

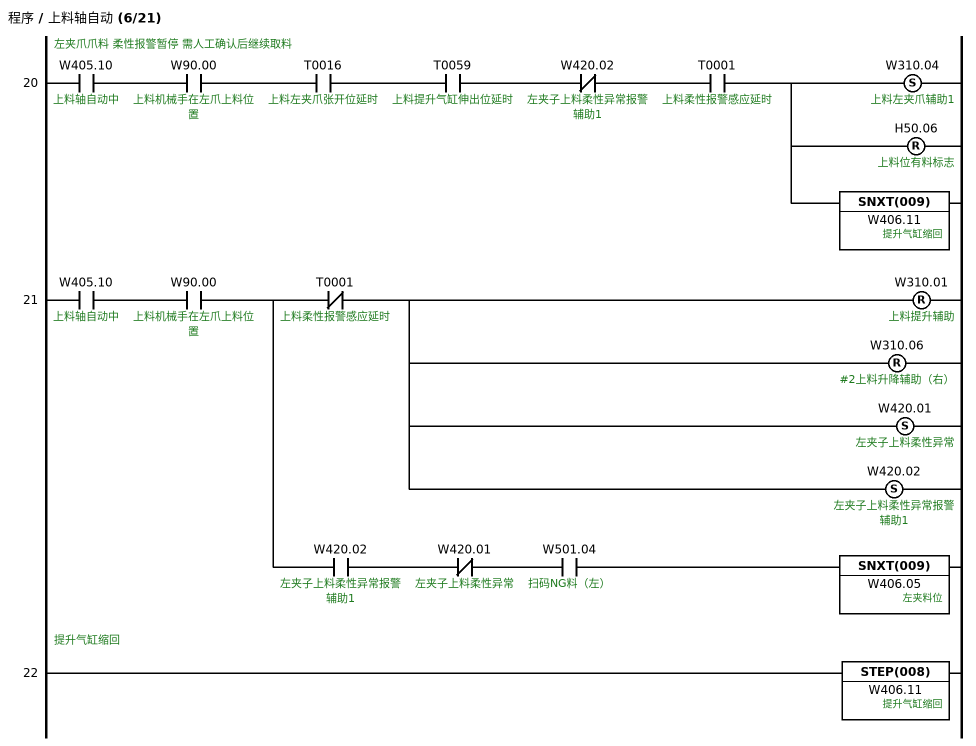
; rung 20: 左夹爪爪料 柔性报警暂停 需人工确认后继续取料
LD W405.10  ; 上料轴自动中
AND W90.00  ; 上料机械手在左爪上料位置
AND T0016  ; 上料左夹爪张开位延时
AND T0059  ; 上料提升气缸伸出位延时
ANDNOT W420.02  ; 左夹子上料柔性异常报警辅助1
AND T0001  ; 上料柔性报警感应延时
SET W310.04  ; 上料左夹爪辅助1
RSET H50.06  ; 上料位有料标志
SNXT(009) W406.11  ; 提升气缸缩回
; rung 21
LD W405.10  ; 上料轴自动中
AND W90.00  ; 上料机械手在左爪上料位置
OUT TR0
ANDNOT T0001  ; 上料柔性报警感应延时
RSET W310.01  ; 上料提升辅助
RSET W310.06  ; #2上料升降辅助（右）
SET W420.01  ; 左夹子上料柔性异常
SET W420.02  ; 左夹子上料柔性异常报警辅助1
LD TR0
AND W420.02  ; 左夹子上料柔性异常报警辅助1
ANDNOT W420.01  ; 左夹子上料柔性异常
AND W501.04  ; 扫码NG料（左）
SNXT(009) W406.05  ; 左夹料位
; rung 22: 提升气缸缩回
STEP(008) W406.11  ; 提升气缸缩回

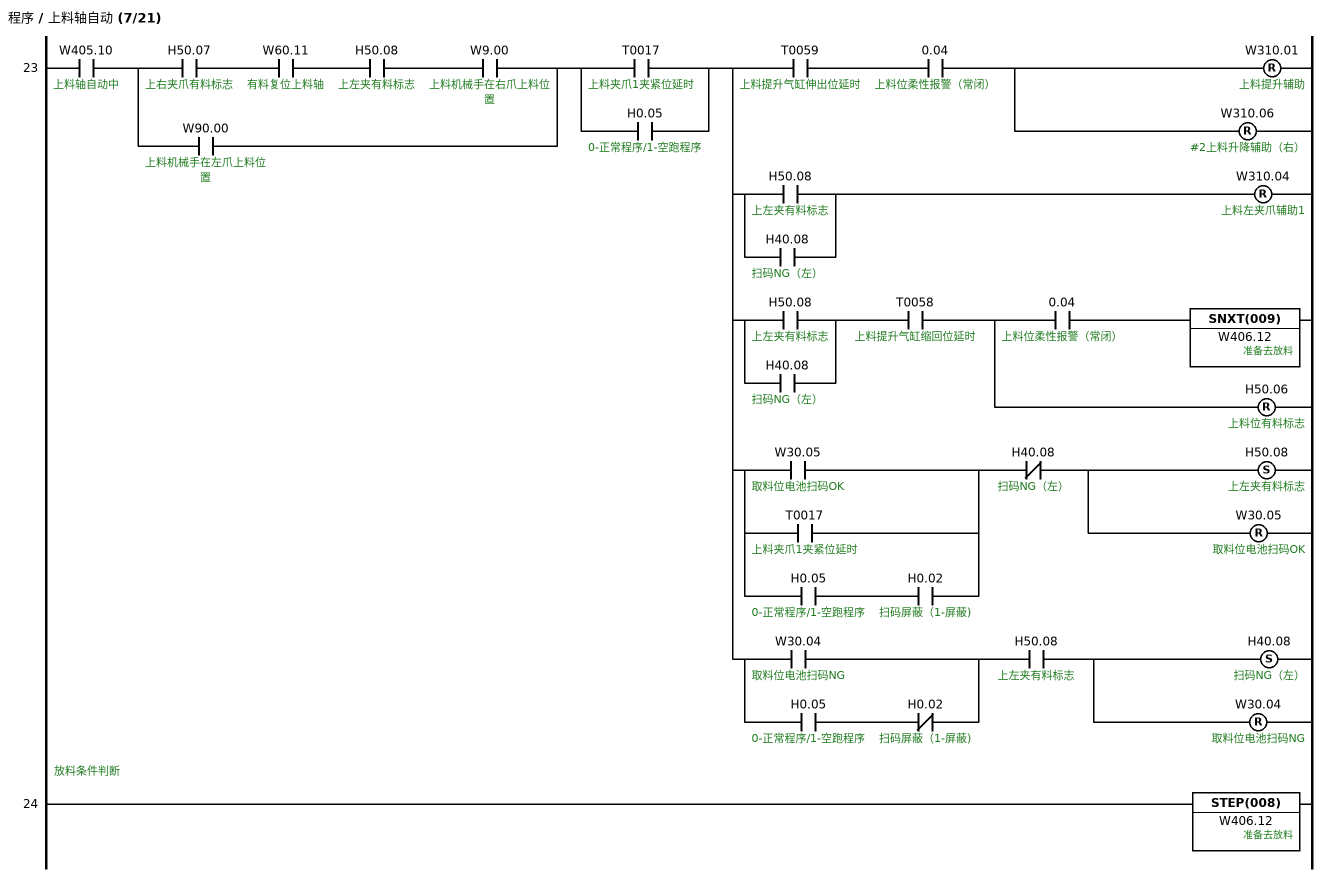
; rung 23
LD W405.10  ; 上料轴自动中
LD H50.07  ; 上右夹爪有料标志
AND W60.11  ; 有料复位上料轴
AND H50.08  ; 上左夹有料标志
AND W9.00  ; 上料机械手在右爪上料位置
OR W90.00  ; 上料机械手在左爪上料位置
ANDLD
LD T0017  ; 上料夹爪1夹紧位延时
OR H0.05  ; 0-正常程序/1-空跑程序
ANDLD
OUT TR0
AND T0059  ; 上料提升气缸伸出位延时
AND 0.04  ; 上料位柔性报警（常闭）
RSET W310.01  ; 上料提升辅助
RSET W310.06  ; #2上料升降辅助（右）
LD TR0
LD H50.08  ; 上左夹有料标志
OR H40.08  ; 扫码NG（左）
ANDLD
RSET W310.04  ; 上料左夹爪辅助1
LD TR0
LD H50.08  ; 上左夹有料标志
OR H40.08  ; 扫码NG（左）
ANDLD
AND T0058  ; 上料提升气缸缩回位延时
OUT TR1
AND 0.04  ; 上料位柔性报警（常闭）
SNXT(009) W406.12  ; 准备去放料
LD TR1
RSET H50.06  ; 上料位有料标志
LD TR0
LD W30.05  ; 取料位电池扫码OK
OR T0017  ; 上料夹爪1夹紧位延时
LD H0.05  ; 0-正常程序/1-空跑程序
AND H0.02  ; 扫码屏蔽（1-屏蔽)
ORLD
ANDLD
ANDNOT H40.08  ; 扫码NG（左）
SET H50.08  ; 上左夹有料标志
RSET W30.05  ; 取料位电池扫码OK
LD TR0
LD W30.04  ; 取料位电池扫码NG
LD H0.05  ; 0-正常程序/1-空跑程序
ANDNOT H0.02  ; 扫码屏蔽（1-屏蔽)
ORLD
ANDLD
AND H50.08  ; 上左夹有料标志
SET H40.08  ; 扫码NG（左）
RSET W30.04  ; 取料位电池扫码NG
; rung 24: 放料条件判断
STEP(008) W406.12  ; 准备去放料

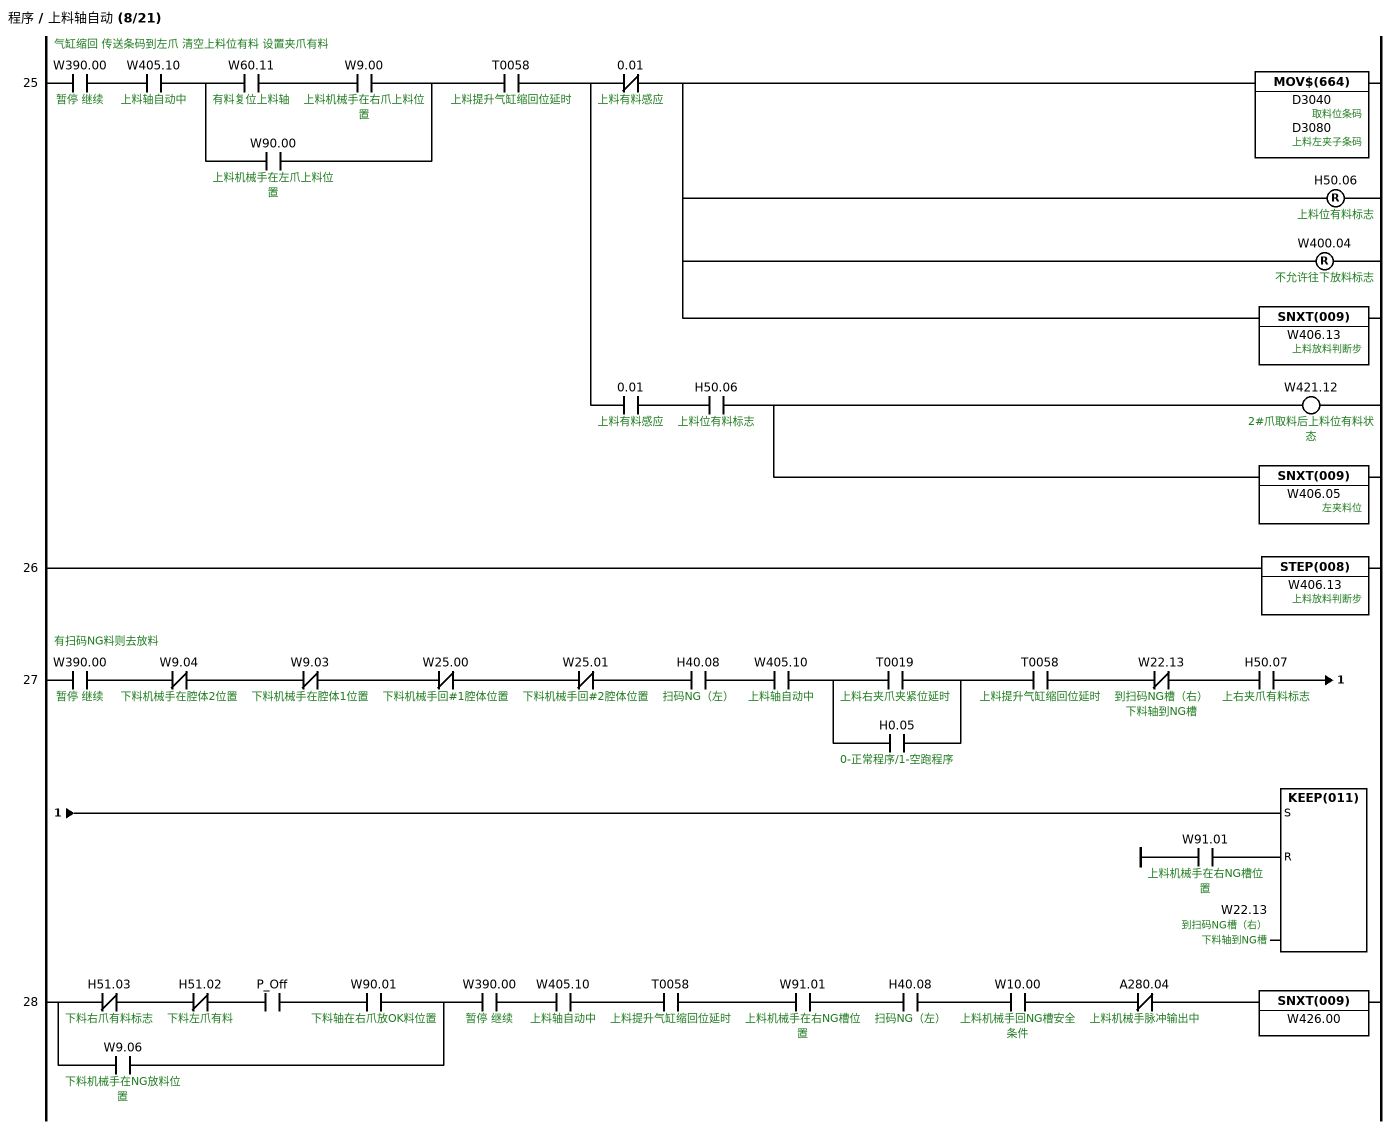
; rung 25: 气缸缩回 传送条码到左爪 清空上料位有料 设置夹爪有料
LD W390.00  ; 暂停 继续
AND W405.10  ; 上料轴自动中
LD W60.11  ; 有料复位上料轴
AND W9.00  ; 上料机械手在右爪上料位置
OR W90.00  ; 上料机械手在左爪上料位置
ANDLD
AND T0058  ; 上料提升气缸缩回位延时
OUT TR0
ANDNOT 0.01  ; 上料有料感应
MOV$(664) D3040 D3080  ; 取料位条码, 上料左夹子条码
RSET H50.06  ; 上料位有料标志
RSET W400.04  ; 不允许往下放料标志
SNXT(009) W406.13  ; 上料放料判断步
LD TR0
AND 0.01  ; 上料有料感应
AND H50.06  ; 上料位有料标志
OUT W421.12  ; 2#爪取料后上料位有料状态
SNXT(009) W406.05  ; 左夹料位
; rung 26
STEP(008) W406.13  ; 上料放料判断步
; rung 27: 有扫码NG料则去放料
LD W390.00  ; 暂停 继续
ANDNOT W9.04  ; 下料机械手在腔体2位置
ANDNOT W9.03  ; 下料机械手在腔体1位置
ANDNOT W25.00  ; 下料机械手回#1腔体位置
ANDNOT W25.01  ; 下料机械手回#2腔体位置
AND H40.08  ; 扫码NG（左）
AND W405.10  ; 上料轴自动中
LD T0019  ; 上料右夹爪夹紧位延时
OR H0.05  ; 0-正常程序/1-空跑程序
ANDLD
AND T0058  ; 上料提升气缸缩回位延时
ANDNOT W22.13  ; 到扫码NG槽（右） 下料轴到NG槽
AND H50.07  ; 上右夹爪有料标志
LD W91.01  ; 上料机械手在右NG槽位置
KEEP(011) W22.13  ; 到扫码NG槽（右） 下料轴到NG槽
; rung 28
LDNOT H51.03  ; 下料右爪有料标志
ANDNOT H51.02  ; 下料左爪有料
AND P_Off
AND W90.01  ; 下料轴在右爪放OK料位置
OR W9.06  ; 下料机械手在NG放料位置
AND W390.00  ; 暂停 继续
AND W405.10  ; 上料轴自动中
AND T0058  ; 上料提升气缸缩回位延时
AND W91.01  ; 上料机械手在右NG槽位置
AND H40.08  ; 扫码NG（左）
AND W10.00  ; 上料机械手回NG槽安全条件
ANDNOT A280.04  ; 上料机械手脉冲输出中
SNXT(009) W426.00

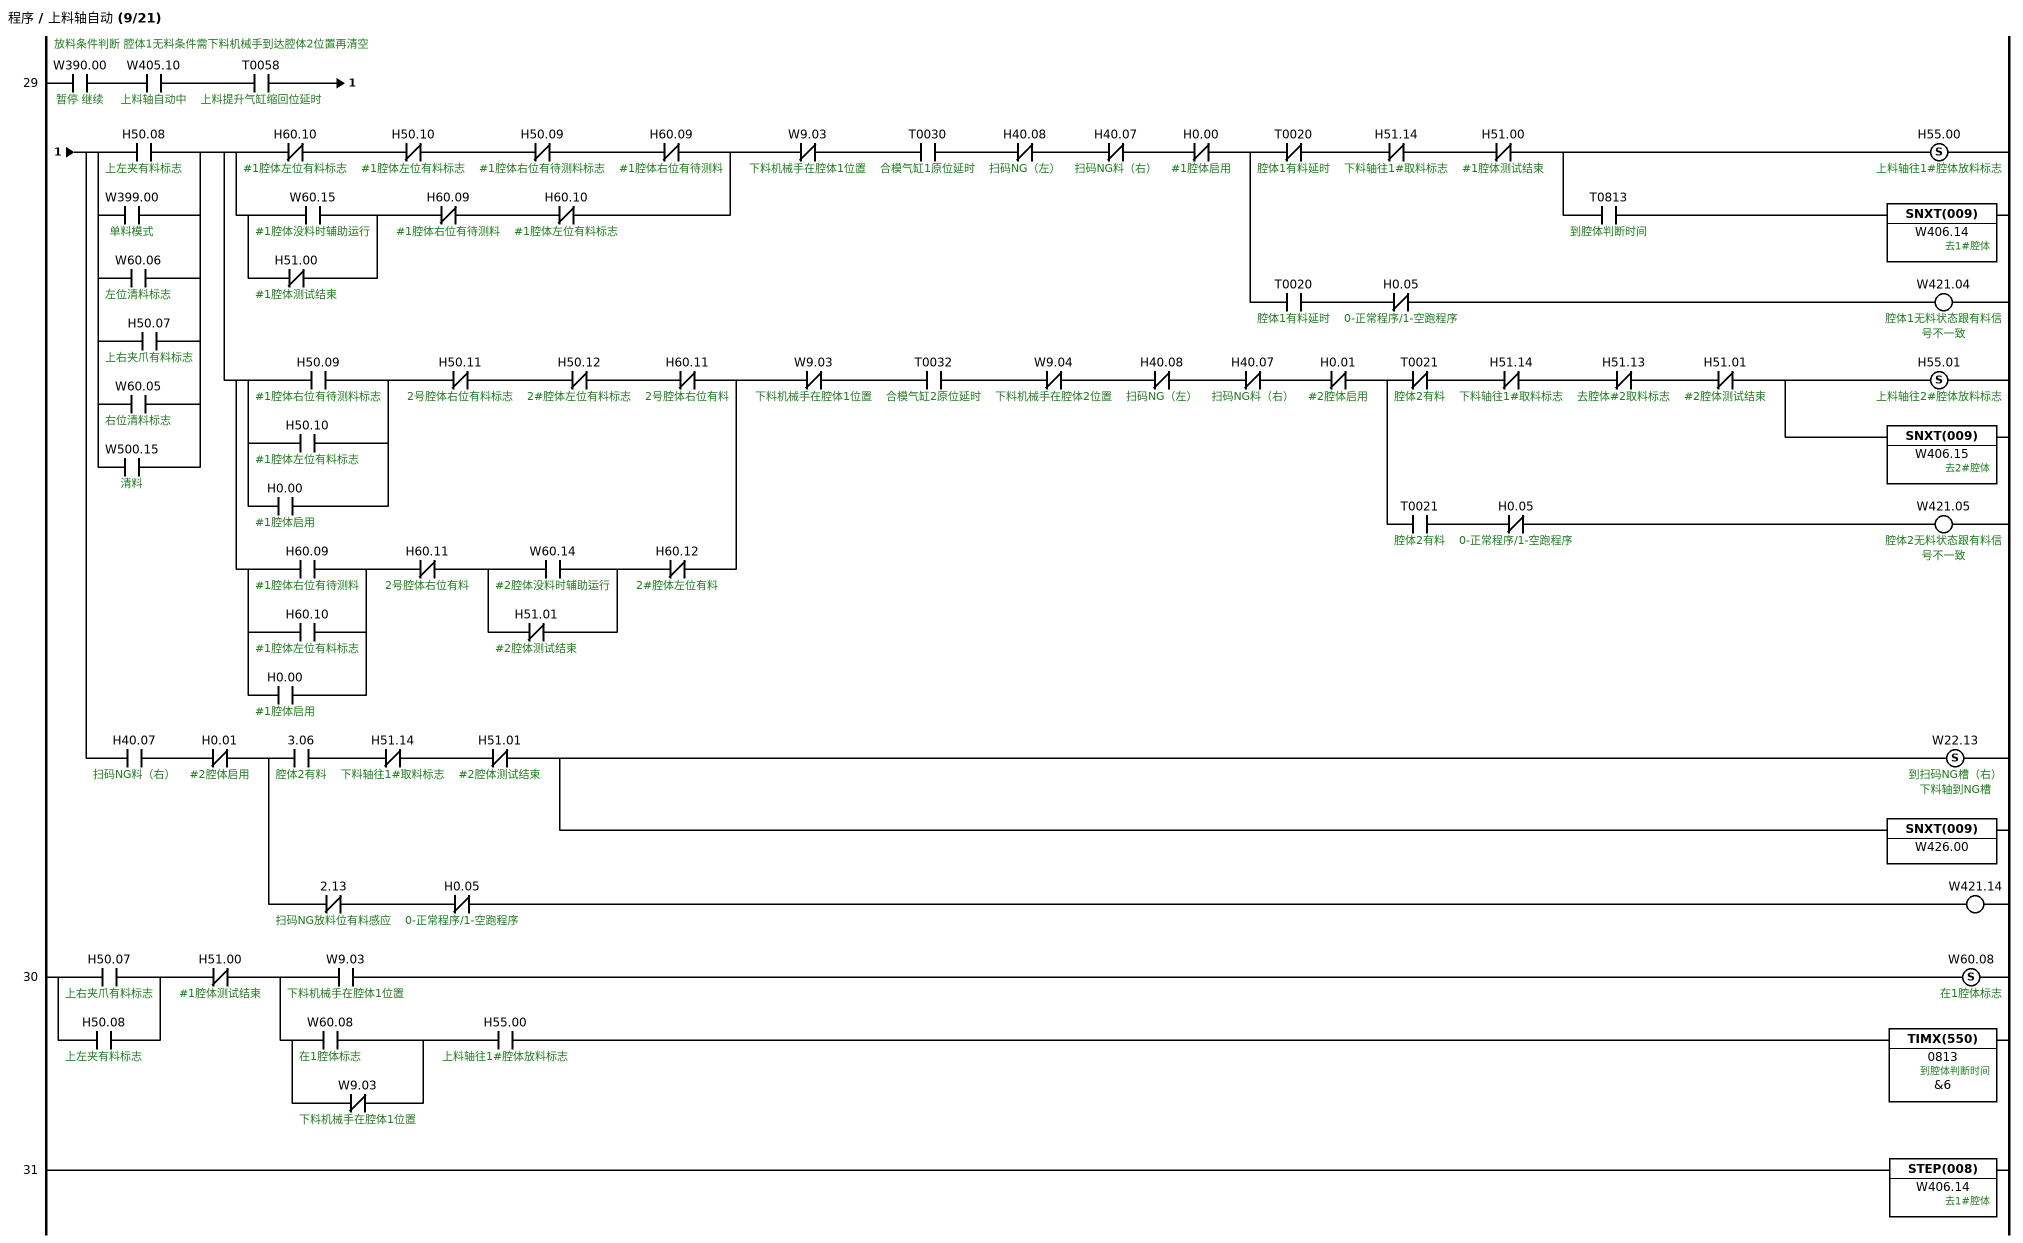
; rung 29: 放料条件判断 腔体1无料条件需下料机械手到达腔体2位置再清空
LD W390.00  ; 暂停 继续
AND W405.10  ; 上料轴自动中
AND T0058  ; 上料提升气缸缩回位延时
OUT TR0
LD H50.08  ; 上左夹有料标志
OR W399.00  ; 单料模式
OR W60.06  ; 左位清料标志
OR H50.07  ; 上右夹爪有料标志
OR W60.05  ; 右位清料标志
OR W500.15  ; 清料
ANDLD
OUT TR1
LDNOT H60.10  ; #1腔体左位有料标志
ANDNOT H50.10  ; #1腔体左位有料标志
ANDNOT H50.09  ; #1腔体右位有待测料标志
ANDNOT H60.09  ; #1腔体右位有待测料
LD W60.15  ; #1腔体没料时辅助运行
ORNOT H51.00  ; #1腔体测试结束
ANDNOT H60.09  ; #1腔体右位有待测料
ANDNOT H60.10  ; #1腔体左位有料标志
ORLD
ANDLD
ANDNOT W9.03  ; 下料机械手在腔体1位置
AND T0030  ; 合模气缸1原位延时
ANDNOT H40.08  ; 扫码NG（左）
ANDNOT H40.07  ; 扫码NG料（右）
ANDNOT H0.00  ; #1腔体启用
OUT TR2
ANDNOT T0020  ; 腔体1有料延时
ANDNOT H51.14  ; 下料轴往1#取料标志
ANDNOT H51.00  ; #1腔体测试结束
SET H55.00  ; 上料轴往1#腔体放料标志
AND T0813  ; 到腔体判断时间
SNXT(009) W406.14  ; 去1#腔体
LD TR2
AND T0020  ; 腔体1有料延时
ANDNOT H0.05  ; 0-正常程序/1-空跑程序
OUT W421.04  ; 腔体1无料状态跟有料信号不一致
LD TR1
LD H50.09  ; #1腔体右位有待测料标志
OR H50.10  ; #1腔体左位有料标志
OR H0.00  ; #1腔体启用
ANDNOT H50.11  ; 2号腔体右位有料标志
ANDNOT H50.12  ; 2#腔体左位有料标志
ANDNOT H60.11  ; 2号腔体右位有料
LD H60.09  ; #1腔体右位有待测料
OR H60.10  ; #1腔体左位有料标志
OR H0.00  ; #1腔体启用
ANDNOT H60.11  ; 2号腔体右位有料
LD W60.14  ; #2腔体没料时辅助运行
ORNOT H51.01  ; #2腔体测试结束
ANDLD
ANDNOT H60.12  ; 2#腔体左位有料
ORLD
ANDLD
ANDNOT W9.03  ; 下料机械手在腔体1位置
AND T0032  ; 合模气缸2原位延时
ANDNOT W9.04  ; 下料机械手在腔体2位置
ANDNOT H40.08  ; 扫码NG（左）
ANDNOT H40.07  ; 扫码NG料（右）
ANDNOT H0.01  ; #2腔体启用
OUT TR1
ANDNOT T0021  ; 腔体2有料
ANDNOT H51.14  ; 下料轴往1#取料标志
ANDNOT H51.13  ; 去腔体#2取料标志
ANDNOT H51.01  ; #2腔体测试结束
SET H55.01  ; 上料轴往2#腔体放料标志
SNXT(009) W406.15  ; 去2#腔体
LD TR1
AND T0021  ; 腔体2有料
ANDNOT H0.05  ; 0-正常程序/1-空跑程序
OUT W421.05  ; 腔体2无料状态跟有料信号不一致
LD TR0
AND H40.07  ; 扫码NG料（右）
ANDNOT H0.01  ; #2腔体启用
OUT TR0
AND 3.06  ; 腔体2有料
ANDNOT H51.14  ; 下料轴往1#取料标志
ANDNOT H51.01  ; #2腔体测试结束
SET W22.13  ; 到扫码NG槽（右） 下料轴到NG槽
SNXT(009) W426.00
LD TR0
ANDNOT 2.13  ; 扫码NG放料位有料感应
ANDNOT H0.05  ; 0-正常程序/1-空跑程序
OUT W421.14
; rung 30
LD H50.07  ; 上右夹爪有料标志
OR H50.08  ; 上左夹有料标志
ANDNOT H51.00  ; #1腔体测试结束
OUT TR0
AND W9.03  ; 下料机械手在腔体1位置
SET W60.08  ; 在1腔体标志
LD TR0
LD W60.08  ; 在1腔体标志
ORNOT W9.03  ; 下料机械手在腔体1位置
ANDLD
AND H55.00  ; 上料轴往1#腔体放料标志
TIMX(550) 0813 &6  ; 到腔体判断时间
; rung 31
STEP(008) W406.14  ; 去1#腔体

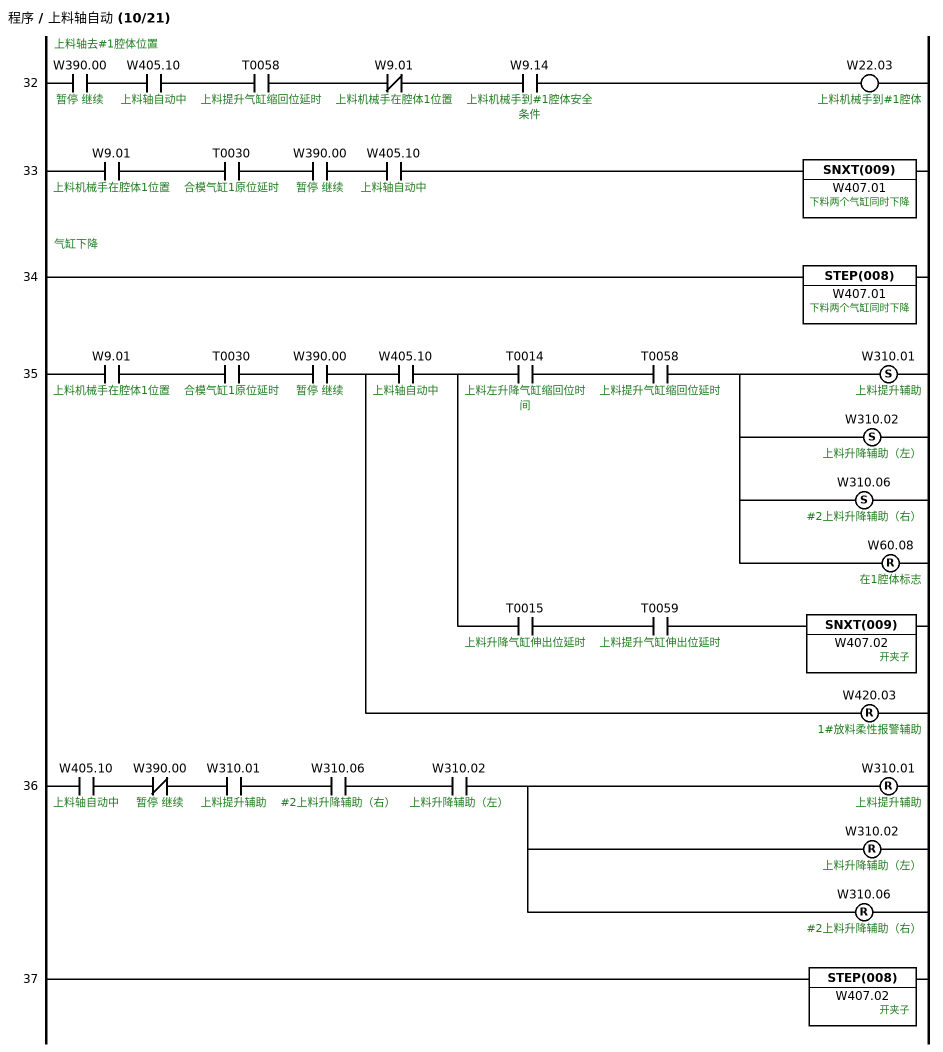
; rung 32: 上料轴去#1腔体位置
LD W390.00  ; 暂停 继续
AND W405.10  ; 上料轴自动中
AND T0058  ; 上料提升气缸缩回位延时
ANDNOT W9.01  ; 上料机械手在腔体1位置
AND W9.14  ; 上料机械手到#1腔体安全条件
OUT W22.03  ; 上料机械手到#1腔体
; rung 33
LD W9.01  ; 上料机械手在腔体1位置
AND T0030  ; 合模气缸1原位延时
AND W390.00  ; 暂停 继续
AND W405.10  ; 上料轴自动中
SNXT(009) W407.01  ; 下料两个气缸同时下降
; rung 34: 气缸下降
STEP(008) W407.01  ; 下料两个气缸同时下降
; rung 35
LD W9.01  ; 上料机械手在腔体1位置
AND T0030  ; 合模气缸1原位延时
AND W390.00  ; 暂停 继续
OUT TR0
AND W405.10  ; 上料轴自动中
OUT TR1
AND T0014  ; 上料左升降气缸缩回位时间
AND T0058  ; 上料提升气缸缩回位延时
SET W310.01  ; 上料提升辅助
SET W310.02  ; 上料升降辅助（左）
SET W310.06  ; #2上料升降辅助（右）
RSET W60.08  ; 在1腔体标志
LD TR1
AND T0015  ; 上料升降气缸伸出位延时
AND T0059  ; 上料提升气缸伸出位延时
SNXT(009) W407.02  ; 开夹子
LD TR0
RSET W420.03  ; 1#放料柔性报警辅助
; rung 36
LD W405.10  ; 上料轴自动中
ANDNOT W390.00  ; 暂停 继续
AND W310.01  ; 上料提升辅助
AND W310.06  ; #2上料升降辅助（右）
AND W310.02  ; 上料升降辅助（左）
RSET W310.01  ; 上料提升辅助
RSET W310.02  ; 上料升降辅助（左）
RSET W310.06  ; #2上料升降辅助（右）
; rung 37
STEP(008) W407.02  ; 开夹子

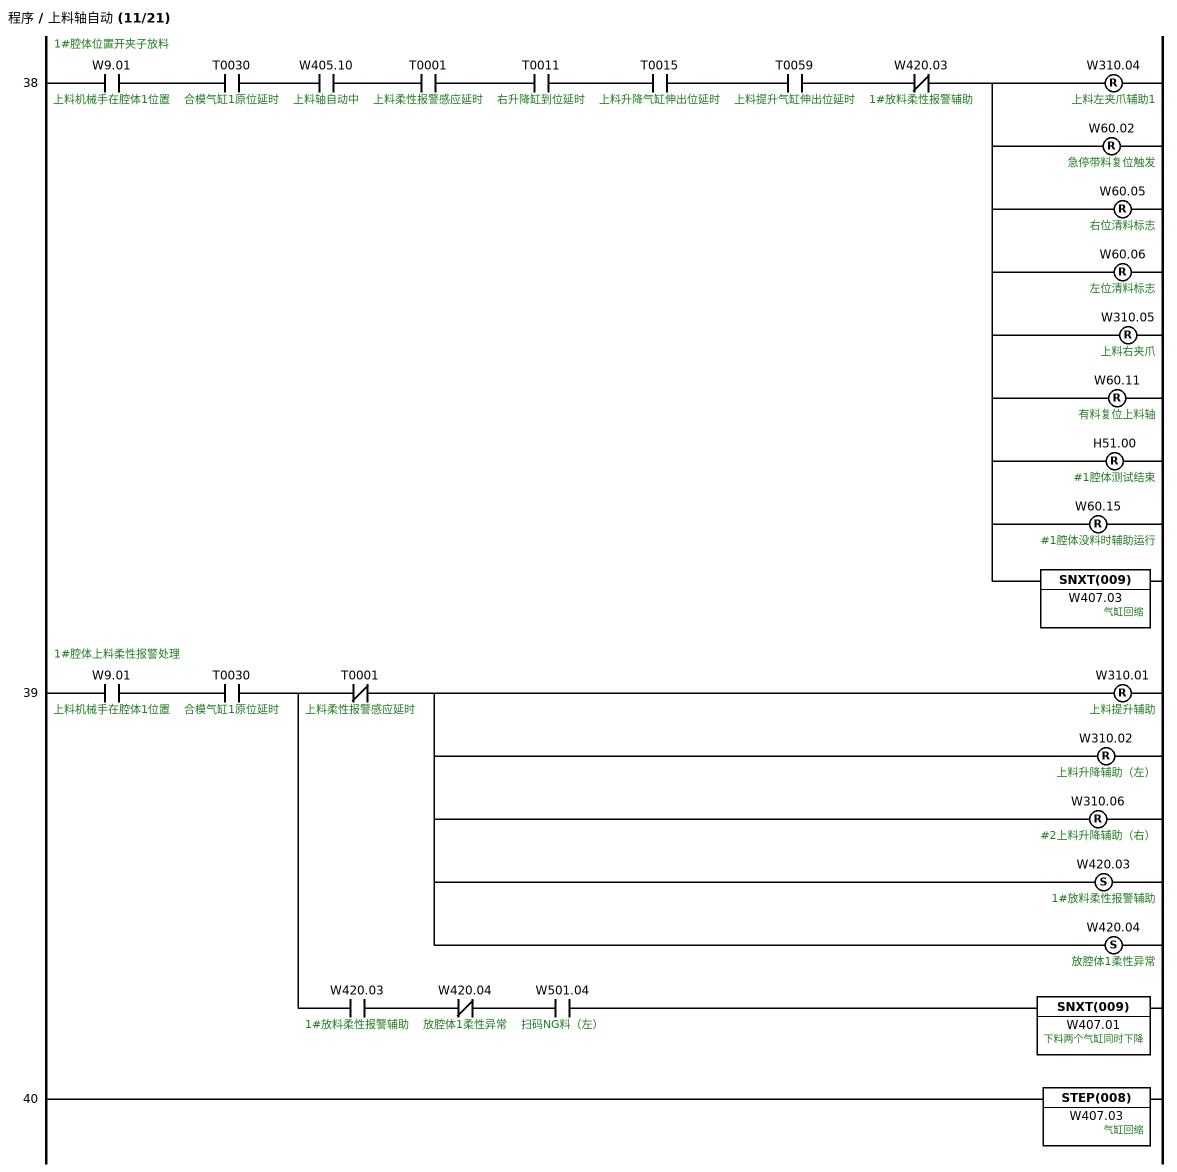
; rung 38: 1#腔体位置开夹子放料
LD W9.01  ; 上料机械手在腔体1位置
AND T0030  ; 合模气缸1原位延时
AND W405.10  ; 上料轴自动中
AND T0001  ; 上料柔性报警感应延时
AND T0011  ; 右升降缸到位延时
AND T0015  ; 上料升降气缸伸出位延时
AND T0059  ; 上料提升气缸伸出位延时
ANDNOT W420.03  ; 1#放料柔性报警辅助
RSET W310.04  ; 上料左夹爪辅助1
RSET W60.02  ; 急停带料复位触发
RSET W60.05  ; 右位清料标志
RSET W60.06  ; 左位清料标志
RSET W310.05  ; 上料右夹爪
RSET W60.11  ; 有料复位上料轴
RSET H51.00  ; #1腔体测试结束
RSET W60.15  ; #1腔体没料时辅助运行
SNXT(009) W407.03  ; 气缸回缩
; rung 39: 1#腔体上料柔性报警处理
LD W9.01  ; 上料机械手在腔体1位置
AND T0030  ; 合模气缸1原位延时
OUT TR0
ANDNOT T0001  ; 上料柔性报警感应延时
RSET W310.01  ; 上料提升辅助
RSET W310.02  ; 上料升降辅助（左）
RSET W310.06  ; #2上料升降辅助（右）
SET W420.03  ; 1#放料柔性报警辅助
SET W420.04  ; 放腔体1柔性异常
LD TR0
AND W420.03  ; 1#放料柔性报警辅助
ANDNOT W420.04  ; 放腔体1柔性异常
AND W501.04  ; 扫码NG料（左）
SNXT(009) W407.01  ; 下料两个气缸同时下降
; rung 40
STEP(008) W407.03  ; 气缸回缩

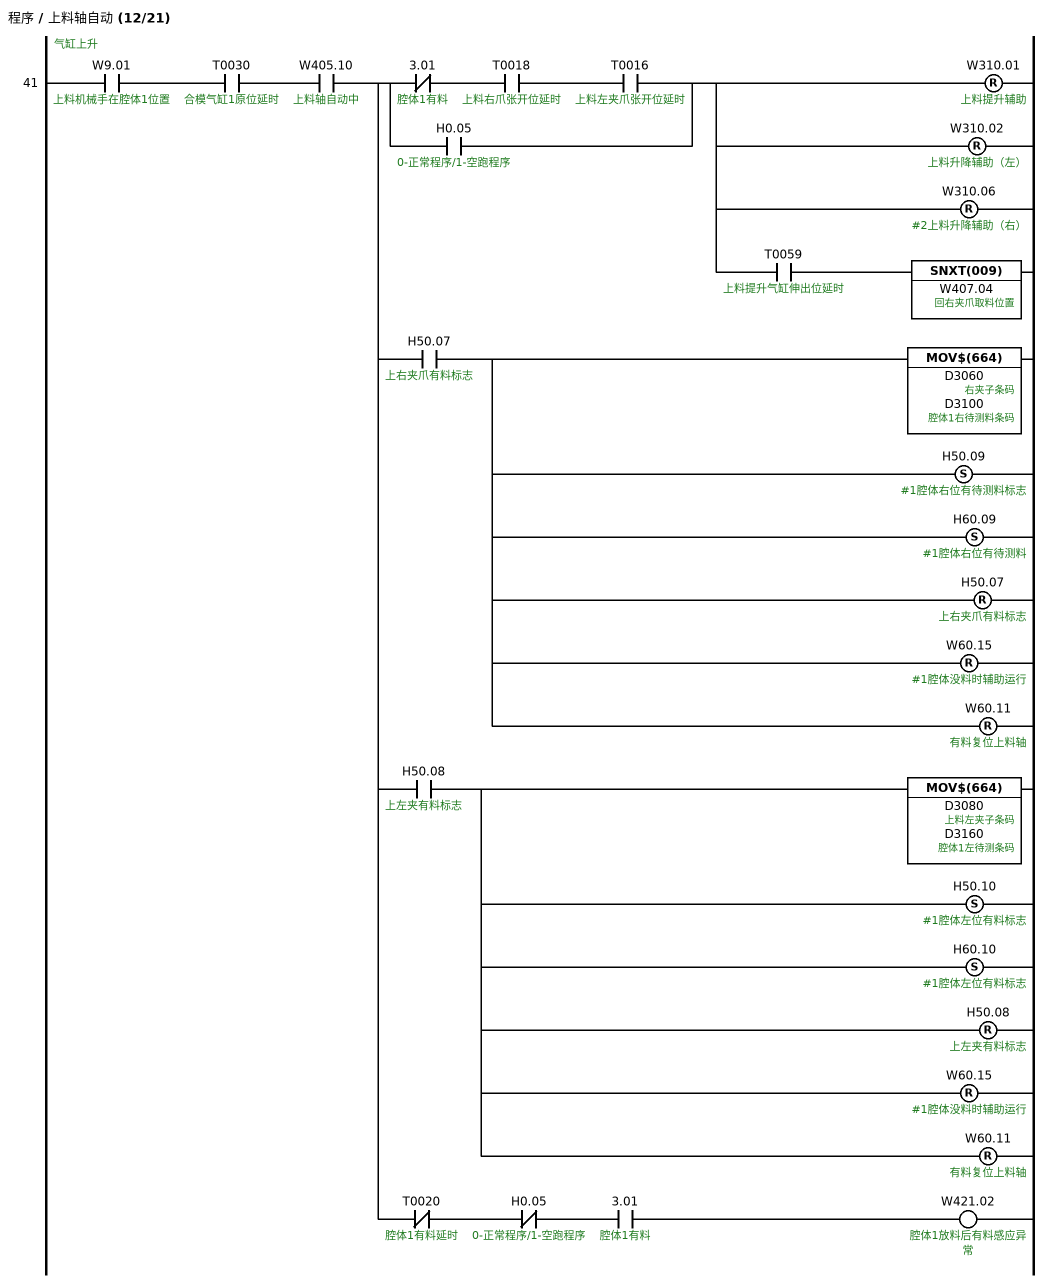
; rung 41: 气缸上升
LD W9.01  ; 上料机械手在腔体1位置
AND T0030  ; 合模气缸1原位延时
AND W405.10  ; 上料轴自动中
OUT TR0
LDNOT 3.01  ; 腔体1有料
AND T0018  ; 上料右爪张开位延时
AND T0016  ; 上料左夹爪张开位延时
OR H0.05  ; 0-正常程序/1-空跑程序
ANDLD
RSET W310.01  ; 上料提升辅助
RSET W310.02  ; 上料升降辅助（左）
RSET W310.06  ; #2上料升降辅助（右）
AND T0059  ; 上料提升气缸伸出位延时
SNXT(009) W407.04  ; 回右夹爪取料位置
LD TR0
AND H50.07  ; 上右夹爪有料标志
MOV$(664) D3060 D3100  ; 右夹子条码, 腔体1右待测料条码
SET H50.09  ; #1腔体右位有待测料标志
SET H60.09  ; #1腔体右位有待测料
RSET H50.07  ; 上右夹爪有料标志
RSET W60.15  ; #1腔体没料时辅助运行
RSET W60.11  ; 有料复位上料轴
LD TR0
AND H50.08  ; 上左夹有料标志
MOV$(664) D3080 D3160  ; 上料左夹子条码, 腔体1左待测条码
SET H50.10  ; #1腔体左位有料标志
SET H60.10  ; #1腔体左位有料标志
RSET H50.08  ; 上左夹有料标志
RSET W60.15  ; #1腔体没料时辅助运行
RSET W60.11  ; 有料复位上料轴
LD TR0
ANDNOT T0020  ; 腔体1有料延时
ANDNOT H0.05  ; 0-正常程序/1-空跑程序
AND 3.01  ; 腔体1有料
OUT W421.02  ; 腔体1放料后有料感应异常

